Yaskawa INFORM job: DEMO_ROOF_UPPER_0625_3PAINT_48.JBI

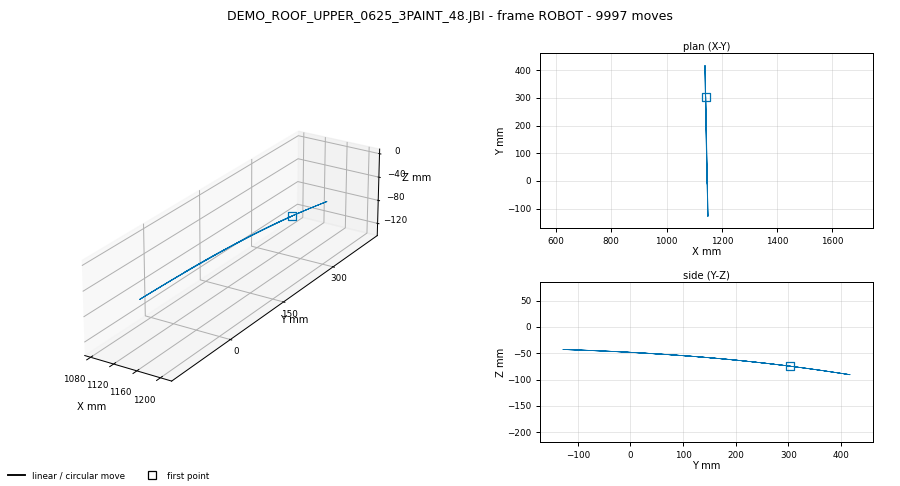
[picture p0: tool path of DEMO_ROOF_UPPER_0625_3PAINT_48.JBI in frame ROBOT, 9997 of 9997 moves have a stored position in this frame; points joined in program order, loops and branches not executed]
/JOB
//NAME DEMO_ROOF_UPPER_0625_3PAINT48
//POS
///NPOS 9997,0,0,0,0,0
///TOOL 0
///USER 0
///POSTYPE ROBOT
///RECTAN
///RCONF 1,0,0,0,0,0,0,0,0,0,0,0,0,0,0,0,0,0,0,0,0,0,0,0
C00000=1141.812,303.776,-74.472,-176.975,8.653,148.834
C00001=1141.816,303.528,-74.441,-176.978,8.649,148.834
C00002=1141.820,303.279,-74.410,-176.981,8.646,148.834
C00003=1141.824,303.032,-74.378,-176.983,8.643,148.834
C00004=1141.829,302.783,-74.347,-176.986,8.639,148.834
C00005=1141.833,302.536,-74.316,-176.989,8.636,148.834
C00006=1141.837,302.287,-74.285,-176.991,8.632,148.834
C00007=1141.841,302.040,-74.253,-176.994,8.628,148.833
C00008=1141.845,301.791,-74.222,-176.997,8.625,148.833
C00009=1141.849,301.544,-74.192,-177.000,8.621,148.833
C00010=1141.853,301.296,-74.160,-177.002,8.618,148.833
C00011=1141.857,301.048,-74.129,-177.005,8.615,148.833
C00012=1141.862,300.800,-74.099,-177.008,8.611,148.833
C00013=1141.866,300.552,-74.067,-177.010,8.608,148.833
C00014=1141.870,300.304,-74.036,-177.012,8.605,148.833
C00015=1141.874,300.055,-74.005,-177.016,8.601,148.833
C00016=1141.879,299.808,-73.973,-177.018,8.597,148.832
C00017=1141.883,299.559,-73.942,-177.020,8.594,148.832
C00018=1141.886,299.311,-73.912,-177.024,8.590,148.832
C00019=1141.891,299.063,-73.881,-177.026,8.587,148.832
C00020=1141.895,298.815,-73.849,-177.028,8.584,148.832
C00021=1141.899,298.567,-73.819,-177.032,8.580,148.832
C00022=1141.904,298.320,-73.788,-177.034,8.577,148.832
C00023=1141.907,298.071,-73.757,-177.036,8.574,148.832
C00024=1141.912,297.823,-73.727,-177.039,8.571,148.832
C00025=1141.916,297.575,-73.695,-177.042,8.567,148.831
C00026=1141.921,297.327,-73.665,-177.045,8.564,148.831
C00027=1141.925,297.079,-73.633,-177.047,8.560,148.831
C00028=1141.928,296.831,-73.603,-177.050,8.556,148.831
C00029=1141.933,296.583,-73.572,-177.053,8.553,148.831
C00030=1141.937,296.335,-73.541,-177.055,8.550,148.831
C00031=1141.941,296.087,-73.511,-177.058,8.546,148.831
C00032=1141.945,295.839,-73.480,-177.061,8.543,148.831
C00033=1141.950,295.591,-73.449,-177.063,8.540,148.831
C00034=1141.954,295.342,-73.418,-177.067,8.536,148.831
C00035=1141.958,295.094,-73.388,-177.069,8.533,148.830
C00036=1141.962,294.846,-73.357,-177.071,8.530,148.830
C00037=1141.966,294.598,-73.326,-177.074,8.527,148.830
C00038=1141.970,294.350,-73.296,-177.077,8.523,148.830
C00039=1141.975,294.102,-73.265,-177.080,8.520,148.830
C00040=1141.979,293.855,-73.235,-177.082,8.516,148.830
C00041=1141.983,293.606,-73.204,-177.085,8.512,148.830
C00042=1141.987,293.358,-73.173,-177.088,8.509,148.830
C00043=1141.991,293.110,-73.143,-177.090,8.506,148.830
C00044=1141.996,292.861,-73.112,-177.094,8.502,148.830
C00045=1141.999,292.613,-73.082,-177.096,8.499,148.829
C00046=1142.004,292.365,-73.051,-177.098,8.496,148.829
C00047=1142.009,292.117,-73.021,-177.101,8.493,148.829
C00048=1142.012,291.869,-72.990,-177.104,8.489,148.829
C00049=1142.017,291.621,-72.959,-177.107,8.486,148.829
C00050=1142.021,291.373,-72.930,-177.109,8.483,148.829
C00051=1142.025,291.125,-72.899,-177.112,8.480,148.829
C00052=1142.029,290.877,-72.869,-177.115,8.476,148.829
C00053=1142.033,290.629,-72.838,-177.118,8.473,148.829
C00054=1142.037,290.380,-72.808,-177.120,8.470,148.829
C00055=1142.042,290.132,-72.778,-177.123,8.466,148.829
C00056=1142.046,289.885,-72.747,-177.126,8.463,148.828
C00057=1142.051,289.636,-72.717,-177.128,8.459,148.828
C00058=1142.054,289.388,-72.687,-177.131,8.456,148.828
C00059=1142.059,289.140,-72.656,-177.134,8.452,148.828
C00060=1142.063,288.892,-72.627,-177.136,8.449,148.828
C00061=1142.067,288.644,-72.596,-177.139,8.446,148.828
C00062=1142.071,288.396,-72.566,-177.142,8.443,148.828
C00063=1142.076,288.147,-72.536,-177.144,8.439,148.828
C00064=1142.080,287.899,-72.505,-177.147,8.436,148.828
C00065=1142.084,287.624,-72.472,-177.150,8.432,148.828
C00066=1142.089,287.348,-72.438,-177.153,8.429,148.828
C00067=1142.094,287.073,-72.405,-177.156,8.425,148.828
C00068=1142.098,286.797,-72.372,-177.159,8.421,148.828
C00069=1142.103,286.549,-72.341,-177.162,8.418,148.828
C00070=1142.107,286.301,-72.312,-177.164,8.415,148.827
C00071=1142.111,286.053,-72.282,-177.167,8.412,148.827
C00072=1142.116,285.805,-72.252,-177.170,8.408,148.827
C00073=1142.120,285.557,-72.221,-177.173,8.405,148.827
C00074=1142.124,285.309,-72.192,-177.175,8.402,148.827
C00075=1142.129,285.061,-72.161,-177.178,8.399,148.827
C00076=1142.132,284.812,-72.131,-177.181,8.395,148.827
C00077=1142.136,284.563,-72.102,-177.184,8.392,148.827
C00078=1142.141,284.316,-72.071,-177.186,8.389,148.827
C00079=1142.145,284.067,-72.042,-177.189,8.386,148.827
C00080=1142.149,283.820,-72.011,-177.192,8.382,148.827
C00081=1142.154,283.571,-71.981,-177.194,8.379,148.827
C00082=1142.158,283.323,-71.952,-177.197,8.376,148.827
C00083=1142.162,283.075,-71.922,-177.200,8.373,148.827
C00084=1142.166,282.827,-71.892,-177.202,8.370,148.827
C00085=1142.171,282.578,-71.862,-177.205,8.366,148.826
C00086=1142.175,282.330,-71.833,-177.208,8.363,148.827
C00087=1142.179,282.082,-71.803,-177.210,8.359,148.826
C00088=1142.183,281.834,-71.773,-177.213,8.356,148.826
C00089=1142.187,281.586,-71.744,-177.217,8.353,148.826
C00090=1142.192,281.337,-71.714,-177.219,8.349,148.826
C00091=1142.196,281.090,-71.684,-177.222,8.347,148.826
C00092=1142.200,280.841,-71.654,-177.224,8.343,148.826
C00093=1142.205,280.593,-71.625,-177.227,8.340,148.826
C00094=1142.209,280.345,-71.595,-177.230,8.336,148.826
C00095=1142.213,280.097,-71.566,-177.233,8.333,148.826
C00096=1142.218,279.848,-71.536,-177.235,8.330,148.826
C00097=1142.222,279.600,-71.506,-177.238,8.327,148.826
C00098=1142.226,279.352,-71.476,-177.240,8.324,148.826
C00099=1142.230,279.104,-71.447,-177.244,8.320,148.826
C00100=1142.234,278.855,-71.417,-177.246,8.317,148.826
C00101=1142.239,278.607,-71.388,-177.249,8.314,148.826
C00102=1142.243,278.359,-71.358,-177.251,8.311,148.826
C00103=1142.247,278.111,-71.329,-177.254,8.308,148.826
C00104=1142.252,277.863,-71.300,-177.257,8.304,148.826
C00105=1142.256,277.615,-71.270,-177.260,8.301,148.826
C00106=1142.260,277.367,-71.241,-177.263,8.298,148.826
C00107=1142.264,277.118,-71.211,-177.265,8.295,148.826
C00108=1142.268,276.870,-71.182,-177.268,8.292,148.826
C00109=1142.273,276.622,-71.152,-177.270,8.289,148.826
C00110=1142.277,276.374,-71.123,-177.273,8.285,148.825
C00111=1142.281,276.125,-71.094,-177.276,8.282,148.825
C00112=1142.285,275.877,-71.064,-177.279,8.279,148.826
C00113=1142.290,275.628,-71.035,-177.281,8.276,148.825
C00114=1142.294,275.381,-71.006,-177.284,8.273,148.825
C00115=1142.299,275.132,-70.977,-177.287,8.270,148.825
C00116=1142.303,274.884,-70.947,-177.290,8.266,148.825
C00117=1142.307,274.636,-70.918,-177.293,8.263,148.825
C00118=1142.311,274.387,-70.888,-177.295,8.260,148.825
C00119=1142.315,274.139,-70.859,-177.298,8.257,148.825
C00120=1142.320,273.890,-70.830,-177.300,8.254,148.825
C00121=1142.325,273.643,-70.801,-177.303,8.251,148.825
C00122=1142.329,273.394,-70.772,-177.306,8.247,148.825
C00123=1142.332,273.147,-70.743,-177.309,8.244,148.825
C00124=1142.337,272.898,-70.714,-177.312,8.241,148.825
C00125=1142.341,272.649,-70.685,-177.314,8.238,148.825
C00126=1142.345,272.401,-70.655,-177.317,8.235,148.825
C00127=1142.350,272.153,-70.627,-177.320,8.232,148.825
C00128=1142.354,271.905,-70.597,-177.323,8.228,148.825
C00129=1142.358,271.656,-70.568,-177.325,8.225,148.825
C00130=1142.362,271.408,-70.540,-177.328,8.222,148.825
C00131=1142.367,271.160,-70.511,-177.331,8.219,148.825
C00132=1142.371,270.912,-70.481,-177.333,8.216,148.825
C00133=1142.376,270.663,-70.453,-177.336,8.213,148.825
C00134=1142.380,270.415,-70.423,-177.339,8.210,148.825
C00135=1142.383,270.167,-70.394,-177.342,8.206,148.825
C00136=1142.388,269.919,-70.366,-177.345,8.203,148.825
C00137=1142.393,269.670,-70.336,-177.347,8.200,148.825
C00138=1142.397,269.422,-70.308,-177.350,8.197,148.825
C00139=1142.401,269.174,-70.279,-177.353,8.194,148.825
C00140=1142.406,268.925,-70.250,-177.355,8.191,148.825
C00141=1142.410,268.677,-70.221,-177.358,8.188,148.825
C00142=1142.414,268.428,-70.192,-177.361,8.185,148.825
C00143=1142.418,268.181,-70.164,-177.364,8.181,148.825
C00144=1142.423,267.932,-70.135,-177.366,8.178,148.825
C00145=1142.427,267.684,-70.106,-177.369,8.175,148.825
C00146=1142.431,267.436,-70.078,-177.372,8.172,148.825
C00147=1142.436,267.187,-70.049,-177.374,8.169,148.825
C00148=1142.440,266.939,-70.020,-177.377,8.166,148.825
C00149=1142.444,266.691,-69.992,-177.380,8.163,148.825
C00150=1142.449,266.443,-69.962,-177.383,8.160,148.825
C00151=1142.453,266.194,-69.934,-177.386,8.157,148.825
C00152=1142.457,265.946,-69.906,-177.388,8.153,148.825
C00153=1142.462,265.698,-69.876,-177.391,8.150,148.825
C00154=1142.466,265.449,-69.848,-177.394,8.147,148.825
C00155=1142.470,265.201,-69.820,-177.397,8.144,148.825
C00156=1142.475,264.953,-69.790,-177.399,8.141,148.825
C00157=1142.478,264.704,-69.762,-177.402,8.138,148.825
C00158=1142.483,264.456,-69.734,-177.405,8.135,148.825
C00159=1142.488,264.207,-69.705,-177.408,8.132,148.825
C00160=1142.492,263.960,-69.677,-177.410,8.129,148.825
C00161=1142.496,263.711,-69.648,-177.413,8.125,148.825
C00162=1142.500,263.462,-69.620,-177.416,8.122,148.825
C00163=1142.505,263.214,-69.591,-177.419,8.119,148.825
C00164=1142.509,262.965,-69.563,-177.422,8.117,148.825
C00165=1142.514,262.718,-69.534,-177.424,8.114,148.825
C00166=1142.518,262.469,-69.506,-177.427,8.110,148.825
C00167=1142.522,262.220,-69.477,-177.430,8.107,148.825
C00168=1142.526,261.973,-69.450,-177.432,8.104,148.825
C00169=1142.532,261.699,-69.418,-177.436,8.101,148.825
C00170=1142.536,261.425,-69.387,-177.438,8.098,148.825
C00171=1142.541,261.152,-69.355,-177.442,8.094,148.825
C00172=1142.546,260.878,-69.325,-177.445,8.091,148.825
C00173=1142.549,260.630,-69.296,-177.447,8.088,148.825
C00174=1142.554,260.382,-69.268,-177.450,8.085,148.825
C00175=1142.558,260.133,-69.240,-177.453,8.082,148.825
C00176=1142.563,259.885,-69.211,-177.455,8.079,148.826
C00177=1142.567,259.636,-69.183,-177.458,8.076,148.826
C00178=1142.571,259.389,-69.156,-177.462,8.072,148.826
C00179=1142.576,259.140,-69.127,-177.464,8.070,148.826
C00180=1142.580,258.892,-69.099,-177.467,8.066,148.826
C00181=1142.585,258.643,-69.070,-177.469,8.063,148.826
C00182=1142.589,258.395,-69.043,-177.472,8.060,148.826
C00183=1142.593,258.146,-69.014,-177.475,8.058,148.826
C00184=1142.598,257.898,-68.986,-177.478,8.055,148.826
C00185=1142.602,257.649,-68.959,-177.481,8.052,148.826
C00186=1142.606,257.401,-68.931,-177.483,8.049,148.826
C00187=1142.611,257.152,-68.902,-177.486,8.045,148.826
C00188=1142.615,256.904,-68.874,-177.488,8.043,148.826
C00189=1142.619,256.656,-68.846,-177.491,8.040,148.826
C00190=1142.623,256.408,-68.818,-177.494,8.037,148.826
C00191=1142.628,256.159,-68.790,-177.497,8.034,148.826
C00192=1142.632,255.911,-68.763,-177.500,8.031,148.826
C00193=1142.637,255.663,-68.735,-177.502,8.028,148.826
C00194=1142.641,255.414,-68.706,-177.505,8.025,148.826
C00195=1142.646,255.166,-68.678,-177.508,8.022,148.826
C00196=1142.650,254.917,-68.651,-177.510,8.019,148.826
C00197=1142.654,254.669,-68.623,-177.514,8.015,148.826
C00198=1142.658,254.420,-68.595,-177.517,8.012,148.826
C00199=1142.663,254.171,-68.567,-177.519,8.009,148.826
C00200=1142.667,253.924,-68.540,-177.522,8.006,148.826
C00201=1142.671,253.675,-68.511,-177.525,8.003,148.826
C00202=1142.676,253.426,-68.484,-177.528,8.000,148.827
C00203=1142.680,253.179,-68.457,-177.530,7.998,148.827
C00204=1142.685,252.930,-68.428,-177.533,7.995,148.827
C00205=1142.689,252.681,-68.401,-177.536,7.991,148.827
C00206=1142.693,252.433,-68.373,-177.538,7.988,148.827
C00207=1142.697,252.185,-68.345,-177.541,7.986,148.827
C00208=1142.702,251.936,-68.318,-177.544,7.983,148.827
C00209=1142.706,251.688,-68.290,-177.547,7.980,148.827
C00210=1142.711,251.439,-68.263,-177.550,7.977,148.827
C00211=1142.715,251.191,-68.235,-177.552,7.974,148.827
C00212=1142.719,250.942,-68.207,-177.555,7.971,148.827
C00213=1142.724,250.694,-68.179,-177.558,7.968,148.827
C00214=1142.729,250.445,-68.152,-177.561,7.965,148.827
C00215=1142.732,250.197,-68.124,-177.564,7.962,148.827
C00216=1142.737,249.948,-68.097,-177.566,7.959,148.827
C00217=1142.741,249.701,-68.069,-177.569,7.956,148.827
C00218=1142.746,249.451,-68.042,-177.572,7.953,148.827
C00219=1142.750,249.203,-68.014,-177.574,7.950,148.827
C00220=1142.755,248.955,-67.987,-177.577,7.947,148.827
C00221=1142.759,248.706,-67.960,-177.580,7.944,148.827
C00222=1142.763,248.458,-67.931,-177.583,7.941,148.828
C00223=1142.768,248.209,-67.904,-177.585,7.938,148.828
C00224=1142.772,247.961,-67.877,-177.588,7.936,148.828
C00225=1142.777,247.713,-67.850,-177.591,7.933,148.828
C00226=1142.781,247.464,-67.822,-177.594,7.930,148.828
C00227=1142.785,247.215,-67.795,-177.597,7.927,148.828
C00228=1142.790,246.967,-67.767,-177.599,7.924,148.828
C00229=1142.794,246.719,-67.740,-177.602,7.921,148.828
C00230=1142.798,246.470,-67.713,-177.605,7.918,148.828
C00231=1142.803,246.221,-67.686,-177.608,7.915,148.828
C00232=1142.807,245.974,-67.659,-177.611,7.912,148.828
C00233=1142.811,245.725,-67.632,-177.613,7.909,148.828
C00234=1142.815,245.476,-67.604,-177.616,7.906,148.828
C00235=1142.820,245.227,-67.577,-177.619,7.903,148.829
C00236=1142.824,244.980,-67.549,-177.622,7.900,148.829
C00237=1142.829,244.731,-67.522,-177.625,7.898,148.829
C00238=1142.834,244.483,-67.495,-177.627,7.895,148.829
C00239=1142.838,244.234,-67.468,-177.630,7.892,148.829
C00240=1142.842,243.985,-67.441,-177.633,7.889,148.829
C00241=1142.846,243.737,-67.414,-177.635,7.887,148.829
C00242=1142.851,243.488,-67.387,-177.638,7.884,148.829
C00243=1142.855,243.240,-67.359,-177.641,7.881,148.829
C00244=1142.860,242.992,-67.332,-177.643,7.878,148.829
C00245=1142.865,242.743,-67.305,-177.646,7.875,148.829
C00246=1142.868,242.495,-67.278,-177.649,7.872,148.829
C00247=1142.873,242.246,-67.251,-177.652,7.869,148.829
C00248=1142.877,241.998,-67.224,-177.655,7.866,148.830
C00249=1142.882,241.749,-67.197,-177.657,7.863,148.830
C00250=1142.886,241.501,-67.171,-177.660,7.860,148.830
C00251=1142.890,241.252,-67.144,-177.663,7.858,148.830
C00252=1142.895,241.004,-67.117,-177.666,7.855,148.830
C00253=1142.900,240.755,-67.090,-177.669,7.852,148.830
C00254=1142.903,240.506,-67.063,-177.671,7.849,148.830
C00255=1142.908,240.258,-67.036,-177.674,7.846,148.830
C00256=1142.912,240.009,-67.009,-177.677,7.843,148.830
C00257=1142.917,239.761,-66.983,-177.680,7.840,148.830
C00258=1142.921,239.512,-66.956,-177.683,7.837,148.830
C00259=1142.926,239.264,-66.929,-177.685,7.834,148.830
C00260=1142.930,239.015,-66.902,-177.688,7.832,148.831
C00261=1142.935,238.767,-66.875,-177.691,7.829,148.831
C00262=1142.939,238.519,-66.848,-177.694,7.827,148.831
C00263=1142.943,238.270,-66.822,-177.696,7.824,148.831
C00264=1142.948,238.021,-66.795,-177.699,7.821,148.831
C00265=1142.953,237.773,-66.768,-177.702,7.818,148.831
C00266=1142.957,237.525,-66.742,-177.705,7.815,148.831
C00267=1142.961,237.276,-66.715,-177.708,7.812,148.831
C00268=1142.966,237.028,-66.688,-177.710,7.809,148.831
C00269=1142.970,236.779,-66.662,-177.713,7.806,148.831
C00270=1142.975,236.530,-66.635,-177.716,7.803,148.832
C00271=1142.979,236.282,-66.608,-177.719,7.800,148.832
C00272=1142.984,236.033,-66.582,-177.721,7.798,148.832
C00273=1142.988,235.761,-66.552,-177.724,7.794,148.832
C00274=1142.993,235.489,-66.524,-177.728,7.792,148.832
C00275=1142.998,235.218,-66.494,-177.730,7.789,148.832
C00276=1143.003,234.946,-66.466,-177.734,7.785,148.832
C00277=1143.007,234.697,-66.439,-177.736,7.783,148.832
C00278=1143.012,234.448,-66.413,-177.739,7.780,148.832
C00279=1143.016,234.200,-66.386,-177.742,7.777,148.832
C00280=1143.021,233.952,-66.359,-177.744,7.774,148.833
C00281=1143.025,233.703,-66.333,-177.747,7.771,148.833
C00282=1143.030,233.454,-66.306,-177.750,7.769,148.833
C00283=1143.034,233.205,-66.281,-177.753,7.766,148.833
C00284=1143.038,232.957,-66.254,-177.756,7.763,148.833
C00285=1143.043,232.708,-66.228,-177.759,7.760,148.833
C00286=1143.047,232.460,-66.201,-177.762,7.757,148.833
C00287=1143.052,232.211,-66.175,-177.764,7.755,148.833
C00288=1143.055,231.963,-66.149,-177.767,7.752,148.834
C00289=1143.060,231.714,-66.122,-177.769,7.749,148.834
C00290=1143.064,231.465,-66.096,-177.772,7.746,148.834
C00291=1143.069,231.217,-66.070,-177.776,7.744,148.834
C00292=1143.074,230.969,-66.043,-177.778,7.741,148.834
C00293=1143.078,230.720,-66.018,-177.781,7.738,148.834
C00294=1143.083,230.471,-65.991,-177.784,7.735,148.834
C00295=1143.087,230.223,-65.965,-177.786,7.733,148.834
C00296=1143.091,229.974,-65.939,-177.789,7.730,148.834
C00297=1143.096,229.725,-65.912,-177.792,7.727,148.835
C00298=1143.100,229.477,-65.886,-177.795,7.724,148.835
C00299=1143.105,229.228,-65.861,-177.798,7.722,148.835
C00300=1143.110,228.980,-65.834,-177.801,7.719,148.835
C00301=1143.114,228.731,-65.808,-177.803,7.716,148.835
C00302=1143.118,228.482,-65.782,-177.806,7.714,148.835
C00303=1143.122,228.234,-65.756,-177.808,7.711,148.835
C00304=1143.127,227.985,-65.729,-177.811,7.708,148.835
C00305=1143.131,227.736,-65.704,-177.814,7.705,148.835
C00306=1143.136,227.488,-65.678,-177.817,7.702,148.836
C00307=1143.141,227.240,-65.651,-177.820,7.700,148.836
C00308=1143.145,226.991,-65.625,-177.823,7.697,148.836
C00309=1143.149,226.742,-65.600,-177.825,7.694,148.836
C00310=1143.153,226.493,-65.574,-177.828,7.692,148.836
C00311=1143.158,226.245,-65.549,-177.831,7.689,148.836
C00312=1143.163,225.997,-65.522,-177.834,7.686,148.837
C00313=1143.167,225.748,-65.496,-177.837,7.683,148.837
C00314=1143.171,225.499,-65.470,-177.840,7.680,148.837
C00315=1143.176,225.251,-65.445,-177.842,7.678,148.837
C00316=1143.180,225.002,-65.419,-177.845,7.675,148.837
C00317=1143.185,224.753,-65.393,-177.848,7.673,148.837
C00318=1143.189,224.504,-65.367,-177.851,7.670,148.837
C00319=1143.194,224.256,-65.341,-177.853,7.667,148.837
C00320=1143.198,224.007,-65.316,-177.856,7.664,148.838
C00321=1143.202,223.759,-65.289,-177.858,7.662,148.838
C00322=1143.207,223.510,-65.263,-177.861,7.659,148.838
C00323=1143.211,223.262,-65.238,-177.864,7.656,148.838
C00324=1143.216,223.013,-65.212,-177.867,7.653,148.838
C00325=1143.221,222.764,-65.186,-177.870,7.651,148.838
C00326=1143.225,222.515,-65.160,-177.872,7.648,148.838
C00327=1143.230,222.267,-65.135,-177.876,7.646,148.839
C00328=1143.234,222.019,-65.109,-177.878,7.643,148.839
C00329=1143.238,221.769,-65.084,-177.881,7.640,148.839
C00330=1143.243,221.521,-65.059,-177.884,7.637,148.839
C00331=1143.247,221.272,-65.033,-177.886,7.635,148.839
C00332=1143.252,221.023,-65.007,-177.889,7.632,148.839
C00333=1143.257,220.775,-64.982,-177.892,7.630,148.839
C00334=1143.261,220.527,-64.956,-177.895,7.627,148.840
C00335=1143.265,220.278,-64.930,-177.898,7.624,148.840
C00336=1143.270,220.030,-64.905,-177.900,7.622,148.840
C00337=1143.274,219.781,-64.879,-177.903,7.619,148.840
C00338=1143.279,219.531,-64.854,-177.906,7.616,148.840
C00339=1143.283,219.283,-64.829,-177.909,7.613,148.840
C00340=1143.288,219.034,-64.803,-177.912,7.610,148.840
C00341=1143.292,218.786,-64.777,-177.914,7.609,148.841
C00342=1143.297,218.538,-64.752,-177.917,7.606,148.841
C00343=1143.301,218.288,-64.727,-177.920,7.603,148.841
C00344=1143.306,218.040,-64.701,-177.923,7.600,148.841
C00345=1143.310,217.791,-64.676,-177.925,7.598,148.841
C00346=1143.314,217.542,-64.650,-177.928,7.595,148.841
C00347=1143.320,217.294,-64.625,-177.931,7.592,148.842
C00348=1143.323,217.045,-64.600,-177.934,7.589,148.842
C00349=1143.328,216.797,-64.575,-177.937,7.587,148.842
C00350=1143.332,216.548,-64.550,-177.939,7.585,148.842
C00351=1143.337,216.299,-64.524,-177.942,7.582,148.842
C00352=1143.341,216.051,-64.499,-177.945,7.579,148.842
C00353=1143.346,215.801,-64.473,-177.948,7.576,148.843
C00354=1143.351,215.553,-64.448,-177.950,7.574,148.843
C00355=1143.355,215.304,-64.424,-177.953,7.571,148.843
C00356=1143.359,215.056,-64.398,-177.956,7.569,148.843
C00357=1143.364,214.807,-64.373,-177.959,7.566,148.843
C00358=1143.369,214.558,-64.348,-177.962,7.564,148.843
C00359=1143.373,214.310,-64.322,-177.964,7.561,148.843
C00360=1143.378,214.060,-64.297,-177.968,7.558,148.844
C00361=1143.382,213.812,-64.272,-177.970,7.555,148.844
C00362=1143.386,213.563,-64.247,-177.973,7.553,148.844
C00363=1143.391,213.315,-64.222,-177.976,7.551,148.844
C00364=1143.396,213.066,-64.197,-177.979,7.548,148.844
C00365=1143.400,212.818,-64.172,-177.981,7.545,148.844
C00366=1143.404,212.568,-64.147,-177.984,7.543,148.845
C00367=1143.409,212.320,-64.122,-177.987,7.540,148.845
C00368=1143.414,212.071,-64.097,-177.990,7.537,148.845
C00369=1143.418,211.823,-64.072,-177.992,7.535,148.845
C00370=1143.423,211.574,-64.047,-177.995,7.533,148.845
C00371=1143.427,211.325,-64.022,-177.998,7.530,148.846
C00372=1143.431,211.077,-63.997,-178.001,7.527,148.846
C00373=1143.436,210.828,-63.972,-178.004,7.525,148.846
C00374=1143.441,210.580,-63.947,-178.006,7.522,148.846
C00375=1143.444,210.330,-63.922,-178.009,7.519,148.846
C00376=1143.450,210.082,-63.898,-178.012,7.517,148.847
C00377=1143.454,209.811,-63.871,-178.015,7.514,148.847
C00378=1143.459,209.541,-63.844,-178.018,7.511,148.847
C00379=1143.465,209.269,-63.816,-178.021,7.508,148.847
C00380=1143.470,208.999,-63.790,-178.025,7.506,148.847
C00381=1143.474,208.750,-63.765,-178.027,7.504,148.847
C00382=1143.478,208.502,-63.740,-178.030,7.501,148.848
C00383=1143.483,208.253,-63.715,-178.033,7.498,148.848
C00384=1143.487,208.004,-63.691,-178.035,7.496,148.848
C00385=1143.492,207.755,-63.666,-178.038,7.493,148.848
C00386=1143.496,207.507,-63.641,-178.041,7.491,148.848
C00387=1143.501,207.258,-63.616,-178.044,7.488,148.849
C00388=1143.505,207.009,-63.592,-178.046,7.486,148.849
C00389=1143.510,206.760,-63.567,-178.049,7.483,148.849
C00390=1143.515,206.512,-63.542,-178.052,7.480,148.849
C00391=1143.519,206.263,-63.518,-178.054,7.478,148.849
C00392=1143.524,206.014,-63.493,-178.058,7.475,148.850
C00393=1143.528,205.766,-63.468,-178.061,7.473,148.850
C00394=1143.533,205.517,-63.443,-178.063,7.471,148.850
C00395=1143.537,205.268,-63.419,-178.066,7.468,148.850
C00396=1143.542,205.020,-63.395,-178.069,7.465,148.850
C00397=1143.546,204.770,-63.370,-178.071,7.463,148.851
C00398=1143.551,204.522,-63.346,-178.074,7.460,148.851
C00399=1143.556,204.273,-63.322,-178.078,7.458,148.851
C00400=1143.560,204.024,-63.296,-178.080,7.456,148.851
C00401=1143.564,203.775,-63.272,-178.083,7.453,148.851
C00402=1143.569,203.527,-63.248,-178.086,7.450,148.852
C00403=1143.574,203.278,-63.224,-178.088,7.448,148.852
C00404=1143.578,203.029,-63.199,-178.091,7.446,148.852
C00405=1143.583,202.780,-63.175,-178.094,7.443,148.852
C00406=1143.587,202.532,-63.150,-178.096,7.441,148.852
C00407=1143.591,202.283,-63.126,-178.100,7.438,148.853
C00408=1143.596,202.034,-63.101,-178.102,7.435,148.853
C00409=1143.601,201.786,-63.077,-178.105,7.433,148.853
C00410=1143.606,201.537,-63.053,-178.108,7.430,148.853
C00411=1143.610,201.287,-63.029,-178.110,7.428,148.853
C00412=1143.614,201.039,-63.005,-178.113,7.426,148.854
C00413=1143.619,200.790,-62.980,-178.116,7.423,148.854
C00414=1143.624,200.542,-62.956,-178.119,7.421,148.854
C00415=1143.628,200.293,-62.932,-178.122,7.418,148.854
C00416=1143.633,200.044,-62.907,-178.125,7.416,148.854
C00417=1143.637,199.795,-62.884,-178.127,7.414,148.855
C00418=1143.642,199.547,-62.860,-178.130,7.411,148.855
C00419=1143.646,199.297,-62.835,-178.133,7.408,148.855
C00420=1143.651,199.049,-62.810,-178.136,7.406,148.855
C00421=1143.655,198.800,-62.786,-178.139,7.404,148.856
C00422=1143.660,198.551,-62.763,-178.141,7.401,148.856
C00423=1143.665,198.303,-62.738,-178.144,7.399,148.856
C00424=1143.669,198.054,-62.714,-178.147,7.396,148.856
C00425=1143.673,197.804,-62.691,-178.150,7.394,148.856
C00426=1143.678,197.556,-62.666,-178.153,7.391,148.857
C00427=1143.683,197.307,-62.642,-178.155,7.388,148.857
C00428=1143.688,197.058,-62.618,-178.158,7.387,148.857
C00429=1143.692,196.810,-62.594,-178.161,7.384,148.857
C00430=1143.696,196.561,-62.570,-178.164,7.382,148.857
C00431=1143.701,196.312,-62.547,-178.166,7.379,148.858
C00432=1143.706,196.063,-62.522,-178.170,7.377,148.858
C00433=1143.710,195.814,-62.498,-178.172,7.375,148.858
C00434=1143.715,195.565,-62.474,-178.175,7.372,148.858
C00435=1143.719,195.317,-62.450,-178.177,7.370,148.859
C00436=1143.724,195.068,-62.427,-178.181,7.367,148.859
C00437=1143.728,194.820,-62.403,-178.183,7.364,148.859
C00438=1143.732,194.570,-62.379,-178.186,7.363,148.859
C00439=1143.737,194.321,-62.355,-178.189,7.360,148.859
C00440=1143.742,194.072,-62.331,-178.192,7.358,148.860
C00441=1143.747,193.824,-62.307,-178.194,7.355,148.860
C00442=1143.751,193.575,-62.284,-178.197,7.353,148.860
C00443=1143.756,193.326,-62.260,-178.200,7.350,148.860
C00444=1143.760,193.077,-62.236,-178.203,7.348,148.861
C00445=1143.765,192.829,-62.212,-178.205,7.346,148.861
C00446=1143.769,192.580,-62.189,-178.209,7.343,148.861
C00447=1143.774,192.331,-62.165,-178.211,7.341,148.861
C00448=1143.779,192.082,-62.141,-178.214,7.339,148.862
C00449=1143.783,191.834,-62.117,-178.216,7.337,148.862
C00450=1143.788,191.585,-62.094,-178.220,7.334,148.862
C00451=1143.793,191.336,-62.070,-178.223,7.331,148.862
C00452=1143.797,191.087,-62.046,-178.225,7.329,148.863
C00453=1143.802,190.838,-62.023,-178.228,7.326,148.863
C00454=1143.807,190.589,-61.999,-178.231,7.325,148.863
C00455=1143.811,190.340,-61.975,-178.234,7.322,148.863
C00456=1143.815,190.091,-61.951,-178.236,7.320,148.864
C00457=1143.820,189.842,-61.928,-178.239,7.317,148.864
C00458=1143.824,189.593,-61.904,-178.242,7.315,148.864
C00459=1143.828,189.345,-61.881,-178.245,7.313,148.864
C00460=1143.834,189.096,-61.858,-178.248,7.310,148.864
C00461=1143.838,188.847,-61.835,-178.251,7.308,148.865
C00462=1143.843,188.599,-61.811,-178.253,7.305,148.865
C00463=1143.848,188.350,-61.787,-178.256,7.304,148.865
C00464=1143.852,188.101,-61.764,-178.259,7.301,148.865
C00465=1143.857,187.852,-61.741,-178.262,7.299,148.866
C00466=1143.862,187.603,-61.717,-178.264,7.296,148.866
C00467=1143.866,187.354,-61.693,-178.267,7.294,148.866
C00468=1143.871,187.105,-61.670,-178.270,7.291,148.866
C00469=1143.875,186.856,-61.647,-178.273,7.290,148.867
C00470=1143.880,186.607,-61.623,-178.276,7.287,148.867
C00471=1143.884,186.359,-61.600,-178.278,7.285,148.867
C00472=1143.889,186.110,-61.577,-178.281,7.283,148.868
C00473=1143.893,185.861,-61.554,-178.284,7.280,148.868
C00474=1143.898,185.612,-61.530,-178.287,7.278,148.868
C00475=1143.903,185.362,-61.507,-178.290,7.275,148.868
C00476=1143.907,185.114,-61.483,-178.292,7.273,148.869
C00477=1143.911,184.865,-61.460,-178.295,7.270,148.869
C00478=1143.917,184.617,-61.437,-178.298,7.269,148.869
C00479=1143.921,184.368,-61.414,-178.301,7.266,148.869
C00480=1143.926,184.119,-61.391,-178.303,7.264,148.869
C00481=1143.931,183.849,-61.365,-178.307,7.261,148.870
C00482=1143.936,183.580,-61.341,-178.310,7.259,148.870
C00483=1143.941,183.309,-61.316,-178.313,7.256,148.870
C00484=1143.946,183.040,-61.290,-178.315,7.254,148.871
C00485=1143.951,182.790,-61.267,-178.319,7.252,148.871
C00486=1143.955,182.542,-61.245,-178.321,7.250,148.871
C00487=1143.960,182.293,-61.221,-178.324,7.247,148.871
C00488=1143.965,182.044,-61.198,-178.327,7.245,148.872
C00489=1143.968,181.796,-61.175,-178.330,7.242,148.872
C00490=1143.973,181.547,-61.152,-178.332,7.241,148.872
C00491=1143.978,181.298,-61.129,-178.335,7.238,148.872
C00492=1143.982,181.049,-61.106,-178.338,7.236,148.873
C00493=1143.987,180.801,-61.083,-178.341,7.234,148.873
C00494=1143.992,180.551,-61.060,-178.343,7.231,148.873
C00495=1143.996,180.302,-61.037,-178.347,7.229,148.874
C00496=1144.001,180.053,-61.014,-178.349,7.227,148.874
C00497=1144.006,179.804,-60.991,-178.352,7.224,148.874
C00498=1144.010,179.556,-60.968,-178.355,7.223,148.874
C00499=1144.015,179.306,-60.946,-178.358,7.220,148.875
C00500=1144.020,179.057,-60.922,-178.360,7.218,148.875
C00501=1144.024,178.809,-60.900,-178.363,7.216,148.875
C00502=1144.028,178.560,-60.876,-178.366,7.213,148.875
C00503=1144.033,178.311,-60.855,-178.369,7.212,148.876
C00504=1144.038,178.062,-60.831,-178.371,7.209,148.876
C00505=1144.043,177.813,-60.808,-178.374,7.207,148.876
C00506=1144.047,177.564,-60.785,-178.377,7.204,148.877
C00507=1144.052,177.315,-60.763,-178.380,7.202,148.877
C00508=1144.056,177.067,-60.740,-178.383,7.200,148.877
C00509=1144.061,176.818,-60.717,-178.386,7.198,148.878
C00510=1144.065,176.568,-60.695,-178.388,7.195,148.878
C00511=1144.071,176.320,-60.672,-178.391,7.193,148.878
C00512=1144.075,176.071,-60.650,-178.394,7.192,148.878
C00513=1144.079,175.821,-60.626,-178.397,7.189,148.879
C00514=1144.084,175.573,-60.604,-178.399,7.187,148.879
C00515=1144.089,175.324,-60.581,-178.403,7.185,148.879
C00516=1144.093,175.075,-60.558,-178.405,7.182,148.879
C00517=1144.098,174.825,-60.536,-178.408,7.180,148.880
C00518=1144.103,174.577,-60.513,-178.411,7.178,148.880
C00519=1144.108,174.328,-60.491,-178.414,7.175,148.880
C00520=1144.112,174.079,-60.468,-178.416,7.174,148.881
C00521=1144.117,173.830,-60.446,-178.419,7.172,148.881
C00522=1144.121,173.581,-60.423,-178.422,7.169,148.881
C00523=1144.125,173.332,-60.401,-178.425,7.167,148.881
C00524=1144.131,173.084,-60.378,-178.428,7.165,148.882
C00525=1144.135,172.834,-60.356,-178.430,7.163,148.882
C00526=1144.140,172.585,-60.332,-178.433,7.161,148.882
C00527=1144.145,172.337,-60.311,-178.436,7.158,148.883
C00528=1144.149,172.088,-60.287,-178.438,7.156,148.883
C00529=1144.154,171.839,-60.266,-178.442,7.154,148.883
C00530=1144.158,171.590,-60.244,-178.444,7.152,148.884
C00531=1144.163,171.341,-60.220,-178.448,7.149,148.884
C00532=1144.168,171.092,-60.199,-178.450,7.147,148.884
C00533=1144.172,170.843,-60.176,-178.453,7.146,148.884
C00534=1144.177,170.594,-60.154,-178.456,7.143,148.885
C00535=1144.182,170.345,-60.132,-178.458,7.141,148.885
C00536=1144.186,170.096,-60.109,-178.461,7.138,148.885
C00537=1144.191,169.847,-60.087,-178.464,7.137,148.886
C00538=1144.196,169.598,-60.064,-178.466,7.135,148.886
C00539=1144.200,169.349,-60.043,-178.470,7.132,148.886
C00540=1144.205,169.100,-60.019,-178.472,7.130,148.887
C00541=1144.209,168.851,-59.997,-178.476,7.128,148.887
C00542=1144.214,168.602,-59.976,-178.478,7.126,148.887
C00543=1144.219,168.353,-59.954,-178.480,7.124,148.887
C00544=1144.224,168.105,-59.931,-178.484,7.121,148.888
C00545=1144.228,167.855,-59.909,-178.486,7.120,148.888
C00546=1144.233,167.607,-59.887,-178.489,7.118,148.888
C00547=1144.238,167.357,-59.864,-178.492,7.115,148.889
C00548=1144.243,167.108,-59.843,-178.495,7.113,148.889
C00549=1144.247,166.860,-59.820,-178.498,7.111,148.889
C00550=1144.252,166.611,-59.798,-178.500,7.109,148.889
C00551=1144.256,166.362,-59.776,-178.503,7.107,148.890
C00552=1144.262,166.113,-59.754,-178.506,7.105,148.890
C00553=1144.266,165.863,-59.732,-178.508,7.102,148.890
C00554=1144.271,165.615,-59.710,-178.511,7.101,148.891
C00555=1144.275,165.365,-59.688,-178.514,7.098,148.891
C00556=1144.280,165.117,-59.666,-178.517,7.096,148.891
C00557=1144.284,164.868,-59.644,-178.519,7.094,148.892
C00558=1144.289,164.619,-59.621,-178.523,7.092,148.892
C00559=1144.294,164.370,-59.599,-178.525,7.090,148.892
C00560=1144.299,164.121,-59.578,-178.528,7.088,148.893
C00561=1144.303,163.872,-59.556,-178.531,7.086,148.893
C00562=1144.308,163.623,-59.534,-178.534,7.084,148.893
C00563=1144.312,163.374,-59.512,-178.537,7.081,148.894
C00564=1144.317,163.125,-59.490,-178.540,7.080,148.894
C00565=1144.321,162.876,-59.468,-178.542,7.077,148.894
C00566=1144.326,162.627,-59.446,-178.545,7.075,148.894
C00567=1144.330,162.378,-59.424,-178.548,7.073,148.895
C00568=1144.336,162.129,-59.402,-178.551,7.071,148.895
C00569=1144.341,161.880,-59.381,-178.554,7.069,148.896
C00570=1144.345,161.630,-59.359,-178.556,7.067,148.896
C00571=1144.350,161.382,-59.337,-178.559,7.065,148.896
C00572=1144.354,161.132,-59.315,-178.562,7.063,148.896
C00573=1144.359,160.884,-59.294,-178.565,7.061,148.897
C00574=1144.364,160.634,-59.272,-178.567,7.059,148.897
C00575=1144.368,160.386,-59.250,-178.570,7.057,148.897
C00576=1144.373,160.137,-59.228,-178.573,7.055,148.898
C00577=1144.378,159.887,-59.207,-178.576,7.053,148.898
C00578=1144.383,159.638,-59.185,-178.578,7.051,148.899
C00579=1144.388,159.390,-59.164,-178.581,7.048,148.899
C00580=1144.392,159.140,-59.142,-178.584,7.047,148.899
C00581=1144.397,158.892,-59.120,-178.587,7.045,148.899
C00582=1144.401,158.642,-59.098,-178.590,7.042,148.900
C00583=1144.406,158.393,-59.077,-178.593,7.041,148.900
C00584=1144.410,158.145,-59.056,-178.595,7.038,148.900
C00585=1144.416,157.876,-59.032,-178.598,7.036,148.901
C00586=1144.421,157.607,-59.008,-178.601,7.034,148.901
C00587=1144.426,157.338,-58.986,-178.604,7.032,148.901
C00588=1144.431,157.068,-58.962,-178.607,7.029,148.902
C00589=1144.435,156.820,-58.941,-178.610,7.027,148.902
C00590=1144.440,156.571,-58.919,-178.613,7.026,148.903
C00591=1144.445,156.321,-58.898,-178.616,7.024,148.903
C00592=1144.450,156.073,-58.876,-178.618,7.021,148.903
C00593=1144.454,155.823,-58.854,-178.621,7.019,148.903
C00594=1144.459,155.574,-58.833,-178.624,7.018,148.904
C00595=1144.464,155.326,-58.812,-178.627,7.015,148.904
C00596=1144.469,155.076,-58.791,-178.630,7.013,148.905
C00597=1144.473,154.827,-58.769,-178.633,7.012,148.905
C00598=1144.478,154.579,-58.748,-178.635,7.010,148.905
C00599=1144.483,154.329,-58.727,-178.638,7.007,148.905
C00600=1144.487,154.080,-58.705,-178.641,7.005,148.906
C00601=1144.492,153.831,-58.684,-178.643,7.004,148.906
C00602=1144.496,153.582,-58.663,-178.646,7.002,148.907
C00603=1144.501,153.333,-58.642,-178.649,6.999,148.907
C00604=1144.506,153.084,-58.620,-178.652,6.997,148.907
C00605=1144.511,152.835,-58.599,-178.654,6.996,148.907
C00606=1144.516,152.586,-58.577,-178.658,6.993,148.908
C00607=1144.520,152.337,-58.556,-178.660,6.991,148.908
C00608=1144.525,152.088,-58.535,-178.663,6.990,148.909
C00609=1144.530,151.838,-58.513,-178.666,6.988,148.909
C00610=1144.535,151.590,-58.492,-178.669,6.985,148.909
C00611=1144.539,151.341,-58.471,-178.671,6.983,148.910
C00612=1144.544,151.092,-58.450,-178.674,6.982,148.910
C00613=1144.549,150.843,-58.429,-178.677,6.980,148.910
C00614=1144.553,150.593,-58.408,-178.680,6.977,148.911
C00615=1144.558,150.345,-58.386,-178.683,6.976,148.911
C00616=1144.563,150.095,-58.365,-178.686,6.974,148.911
C00617=1144.567,149.846,-58.345,-178.688,6.972,148.912
C00618=1144.572,149.598,-58.323,-178.690,6.970,148.912
C00619=1144.577,149.348,-58.302,-178.694,6.968,148.912
C00620=1144.581,149.099,-58.282,-178.696,6.966,148.913
C00621=1144.586,148.850,-58.260,-178.699,6.964,148.913
C00622=1144.591,148.601,-58.239,-178.702,6.963,148.914
C00623=1144.596,148.352,-58.219,-178.705,6.960,148.914
C00624=1144.601,148.103,-58.198,-178.708,6.958,148.914
C00625=1144.606,147.854,-58.176,-178.711,6.957,148.915
C00626=1144.610,147.604,-58.155,-178.713,6.955,148.915
C00627=1144.615,147.355,-58.134,-178.716,6.952,148.915
C00628=1144.619,147.106,-58.114,-178.719,6.950,148.916
C00629=1144.624,146.858,-58.092,-178.722,6.949,148.916
C00630=1144.629,146.608,-58.071,-178.724,6.947,148.916
C00631=1144.634,146.359,-58.051,-178.727,6.945,148.917
C00632=1144.639,146.110,-58.030,-178.730,6.943,148.917
C00633=1144.643,145.861,-58.010,-178.733,6.941,148.917
C00634=1144.648,145.612,-57.989,-178.736,6.939,148.918
C00635=1144.652,145.363,-57.967,-178.738,6.937,148.918
C00636=1144.657,145.114,-57.946,-178.741,6.935,148.918
C00637=1144.662,144.865,-57.926,-178.744,6.933,148.919
C00638=1144.667,144.615,-57.905,-178.747,6.931,148.919
C00639=1144.671,144.366,-57.884,-178.749,6.929,148.920
C00640=1144.676,144.117,-57.863,-178.752,6.928,148.920
C00641=1144.681,143.868,-57.843,-178.755,6.926,148.920
C00642=1144.686,143.619,-57.822,-178.758,6.924,148.921
C00643=1144.690,143.370,-57.802,-178.761,6.922,148.921
C00644=1144.696,143.121,-57.781,-178.764,6.920,148.921
C00645=1144.700,142.872,-57.760,-178.766,6.918,148.922
C00646=1144.705,142.623,-57.739,-178.769,6.917,148.922
C00647=1144.710,142.374,-57.719,-178.772,6.915,148.923
C00648=1144.714,142.125,-57.699,-178.775,6.912,148.923
C00649=1144.719,141.875,-57.678,-178.777,6.910,148.923
C00650=1144.724,141.626,-57.657,-178.780,6.909,148.924
C00651=1144.729,141.377,-57.636,-178.783,6.907,148.924
C00652=1144.733,141.128,-57.616,-178.785,6.905,148.924
C00653=1144.738,140.879,-57.596,-178.789,6.903,148.925
C00654=1144.743,140.630,-57.575,-178.791,6.901,148.925
C00655=1144.747,140.381,-57.554,-178.794,6.899,148.926
C00656=1144.753,140.132,-57.533,-178.797,6.898,148.926
C00657=1144.757,139.883,-57.513,-178.800,6.896,148.926
C00658=1144.761,139.634,-57.493,-178.802,6.894,148.927
C00659=1144.767,139.385,-57.472,-178.805,6.892,148.927
C00660=1144.771,139.136,-57.451,-178.808,6.890,148.927
C00661=1144.776,138.886,-57.432,-178.811,6.888,148.928
C00662=1144.781,138.637,-57.411,-178.814,6.887,148.928
C00663=1144.785,138.388,-57.390,-178.816,6.885,148.929
C00664=1144.790,138.139,-57.370,-178.819,6.883,148.929
C00665=1144.794,137.890,-57.350,-178.821,6.881,148.929
C00666=1144.800,137.640,-57.329,-178.825,6.879,148.930
C00667=1144.804,137.391,-57.309,-178.827,6.877,148.930
C00668=1144.809,137.142,-57.289,-178.830,6.875,148.930
C00669=1144.814,136.893,-57.268,-178.833,6.873,148.931
C00670=1144.818,136.644,-57.247,-178.836,6.872,148.931
C00671=1144.823,136.395,-57.228,-178.838,6.870,148.932
C00672=1144.828,136.146,-57.208,-178.841,6.868,148.932
C00673=1144.833,135.897,-57.187,-178.844,6.867,148.932
C00674=1144.838,135.647,-57.167,-178.847,6.864,148.933
C00675=1144.842,135.398,-57.147,-178.850,6.862,148.933
C00676=1144.847,135.150,-57.126,-178.852,6.861,148.933
C00677=1144.852,134.900,-57.106,-178.855,6.859,148.934
C00678=1144.857,134.651,-57.086,-178.858,6.857,148.934
C00679=1144.861,134.402,-57.065,-178.861,6.856,148.935
C00680=1144.867,134.153,-57.046,-178.863,6.854,148.935
C00681=1144.871,133.904,-57.025,-178.866,6.852,148.935
C00682=1144.875,133.655,-57.005,-178.869,6.850,148.936
C00683=1144.881,133.405,-56.985,-178.872,6.848,148.936
C00684=1144.885,133.156,-56.964,-178.875,6.846,148.937
C00685=1144.890,132.907,-56.945,-178.877,6.845,148.937
C00686=1144.894,132.658,-56.924,-178.880,6.843,148.937
C00687=1144.900,132.409,-56.905,-178.883,6.841,148.938
C00688=1144.904,132.160,-56.885,-178.886,6.839,148.938
C00689=1144.910,131.891,-56.863,-178.889,6.837,148.939
C00690=1144.915,131.623,-56.841,-178.892,6.835,148.939
C00691=1144.920,131.354,-56.820,-178.894,6.833,148.939
C00692=1144.925,131.085,-56.799,-178.898,6.831,148.940
C00693=1144.930,130.836,-56.778,-178.900,6.829,148.940
C00694=1144.934,130.587,-56.759,-178.903,6.828,148.941
C00695=1144.939,130.338,-56.739,-178.906,6.826,148.941
C00696=1144.944,130.089,-56.719,-178.909,6.824,148.941
C00697=1144.949,129.839,-56.699,-178.911,6.822,148.942
C00698=1144.953,129.590,-56.679,-178.914,6.821,148.942
C00699=1144.959,129.342,-56.660,-178.917,6.819,148.943
C00700=1144.963,129.093,-56.639,-178.920,6.818,148.943
C00701=1144.968,128.843,-56.619,-178.923,6.816,148.944
C00702=1144.973,128.593,-56.599,-178.925,6.814,148.944
C00703=1144.978,128.345,-56.579,-178.928,6.813,148.944
C00704=1144.983,128.095,-56.560,-178.931,6.811,148.945
C00705=1144.987,127.846,-56.539,-178.934,6.808,148.945
C00706=1144.992,127.597,-56.520,-178.937,6.807,148.945
C00707=1144.997,127.348,-56.501,-178.940,6.805,148.946
C00708=1145.002,127.099,-56.481,-178.942,6.803,148.946
C00709=1145.006,126.850,-56.461,-178.945,6.802,148.947
C00710=1145.011,126.600,-56.441,-178.948,6.800,148.947
C00711=1145.016,126.351,-56.422,-178.950,6.798,148.947
C00712=1145.021,126.102,-56.402,-178.953,6.797,148.948
C00713=1145.025,125.853,-56.382,-178.956,6.795,148.948
C00714=1145.031,125.604,-56.363,-178.959,6.793,148.949
C00715=1145.035,125.354,-56.343,-178.961,6.791,148.949
C00716=1145.040,125.105,-56.323,-178.964,6.790,148.949
C00717=1145.045,124.856,-56.303,-178.967,6.788,148.950
C00718=1145.050,124.607,-56.284,-178.969,6.786,148.950
C00719=1145.054,124.358,-56.265,-178.972,6.785,148.951
C00720=1145.059,124.108,-56.245,-178.975,6.783,148.951
C00721=1145.064,123.860,-56.225,-178.978,6.781,148.951
C00722=1145.068,123.610,-56.205,-178.980,6.780,148.952
C00723=1145.073,123.361,-56.186,-178.983,6.778,148.952
C00724=1145.078,123.112,-56.166,-178.986,6.776,148.953
C00725=1145.083,122.862,-56.147,-178.989,6.774,148.953
C00726=1145.088,122.614,-56.128,-178.992,6.772,148.953
C00727=1145.093,122.364,-56.108,-178.995,6.770,148.954
C00728=1145.097,122.115,-56.089,-178.998,6.769,148.954
C00729=1145.103,121.866,-56.069,-179.000,6.767,148.955
C00730=1145.107,121.616,-56.050,-179.003,6.765,148.955
C00731=1145.111,121.368,-56.030,-179.006,6.764,148.956
C00732=1145.116,121.119,-56.011,-179.009,6.762,148.956
C00733=1145.121,120.869,-55.991,-179.011,6.760,148.956
C00734=1145.127,120.620,-55.972,-179.014,6.759,148.957
C00735=1145.131,120.371,-55.953,-179.017,6.757,148.957
C00736=1145.135,120.121,-55.933,-179.020,6.755,148.958
C00737=1145.141,119.873,-55.914,-179.022,6.754,148.958
C00738=1145.145,119.623,-55.894,-179.025,6.752,148.958
C00739=1145.150,119.374,-55.875,-179.028,6.750,148.959
C00740=1145.155,119.125,-55.856,-179.030,6.749,148.959
C00741=1145.160,118.875,-55.837,-179.033,6.747,148.960
C00742=1145.165,118.626,-55.817,-179.036,6.745,148.960
C00743=1145.169,118.377,-55.798,-179.039,6.744,148.961
C00744=1145.174,118.128,-55.779,-179.042,6.742,148.961
C00745=1145.179,117.878,-55.759,-179.045,6.740,148.962
C00746=1145.184,117.630,-55.741,-179.047,6.739,148.962
C00747=1145.189,117.380,-55.721,-179.050,6.737,148.962
C00748=1145.194,117.131,-55.702,-179.053,6.735,148.963
C00749=1145.198,116.882,-55.683,-179.055,6.734,148.963
C00750=1145.204,116.632,-55.664,-179.058,6.732,148.964
C00751=1145.208,116.383,-55.644,-179.061,6.730,148.964
C00752=1145.213,116.134,-55.626,-179.064,6.729,148.964
C00753=1145.218,115.885,-55.606,-179.066,6.727,148.965
C00754=1145.223,115.636,-55.587,-179.070,6.726,148.965
C00755=1145.227,115.386,-55.568,-179.072,6.725,148.966
C00756=1145.233,115.137,-55.549,-179.074,6.723,148.966
C00757=1145.237,114.888,-55.530,-179.077,6.721,148.967
C00758=1145.242,114.639,-55.511,-179.080,6.720,148.967
C00759=1145.247,114.389,-55.492,-179.083,6.718,148.967
C00760=1145.252,114.140,-55.473,-179.085,6.716,148.968
C00761=1145.256,113.891,-55.454,-179.088,6.715,148.968
C00762=1145.261,113.642,-55.435,-179.091,6.713,148.969
C00763=1145.267,113.393,-55.416,-179.093,6.711,148.969
C00764=1145.271,113.143,-55.397,-179.097,6.710,148.970
C00765=1145.276,112.894,-55.378,-179.099,6.708,148.970
C00766=1145.280,112.645,-55.360,-179.102,6.706,148.971
C00767=1145.286,112.396,-55.340,-179.105,6.705,148.971
C00768=1145.290,112.146,-55.321,-179.108,6.703,148.971
C00769=1145.295,111.897,-55.303,-179.110,6.701,148.972
C00770=1145.301,111.648,-55.283,-179.113,6.700,148.972
C00771=1145.305,111.399,-55.264,-179.116,6.698,148.973
C00772=1145.310,111.149,-55.246,-179.118,6.696,148.973
C00773=1145.314,110.900,-55.227,-179.122,6.695,148.974
C00774=1145.319,110.651,-55.209,-179.124,6.693,148.974
C00775=1145.325,110.402,-55.189,-179.127,6.692,148.974
C00776=1145.329,110.152,-55.171,-179.129,6.691,148.975
C00777=1145.334,109.903,-55.152,-179.132,6.689,148.975
C00778=1145.338,109.654,-55.133,-179.135,6.687,148.976
C00779=1145.344,109.405,-55.114,-179.137,6.686,148.976
C00780=1145.348,109.156,-55.095,-179.141,6.684,148.977
C00781=1145.354,108.906,-55.076,-179.143,6.683,148.977
C00782=1145.358,108.657,-55.058,-179.146,6.681,148.977
C00783=1145.363,108.408,-55.040,-179.149,6.679,148.978
C00784=1145.368,108.159,-55.020,-179.152,6.678,148.978
C00785=1145.373,107.909,-55.002,-179.154,6.676,148.979
C00786=1145.377,107.659,-54.984,-179.157,6.674,148.979
C00787=1145.382,107.411,-54.965,-179.160,6.672,148.980
C00788=1145.387,107.161,-54.947,-179.163,6.671,148.980
C00789=1145.392,106.912,-54.927,-179.165,6.670,148.981
C00790=1145.397,106.663,-54.909,-179.168,6.669,148.981
C00791=1145.402,106.414,-54.890,-179.171,6.667,148.981
C00792=1145.407,106.164,-54.871,-179.173,6.665,148.982
C00793=1145.412,105.896,-54.852,-179.176,6.664,148.982
C00794=1145.417,105.627,-54.832,-179.179,6.662,148.983
C00795=1145.422,105.359,-54.812,-179.182,6.661,148.983
C00796=1145.427,105.091,-54.792,-179.185,6.658,148.984
C00797=1145.432,104.841,-54.773,-179.188,6.658,148.984
C00798=1145.437,104.592,-54.755,-179.191,6.656,148.985
C00799=1145.442,104.343,-54.737,-179.193,6.654,148.985
C00800=1145.448,104.094,-54.718,-179.196,6.652,148.986
C00801=1145.452,103.844,-54.700,-179.199,6.651,148.986
C00802=1145.456,103.595,-54.681,-179.202,6.649,148.986
C00803=1145.461,103.346,-54.663,-179.205,6.648,148.987
C00804=1145.466,103.096,-54.644,-179.207,6.646,148.987
C00805=1145.471,102.847,-54.626,-179.210,6.644,148.988
C00806=1145.476,102.598,-54.608,-179.212,6.644,148.988
C00807=1145.481,102.349,-54.590,-179.215,6.642,148.989
C00808=1145.487,102.100,-54.571,-179.218,6.640,148.989
C00809=1145.491,101.850,-54.553,-179.221,6.639,148.990
C00810=1145.495,101.601,-54.534,-179.224,6.637,148.990
C00811=1145.500,101.352,-54.516,-179.226,6.635,148.991
C00812=1145.505,101.103,-54.498,-179.229,6.634,148.991
C00813=1145.510,100.853,-54.479,-179.232,6.632,148.991
C00814=1145.515,100.603,-54.461,-179.234,6.631,148.992
C00815=1145.520,100.354,-54.443,-179.237,6.630,148.992
C00816=1145.525,100.105,-54.425,-179.240,6.628,148.993
C00817=1145.530,99.857,-54.406,-179.243,6.627,148.993
C00818=1145.534,99.607,-54.388,-179.246,6.625,148.994
C00819=1145.539,99.358,-54.370,-179.248,6.623,148.994
C00820=1145.545,99.108,-54.351,-179.251,6.622,148.995
C00821=1145.549,98.859,-54.334,-179.254,6.621,148.995
C00822=1145.554,98.610,-54.316,-179.256,6.619,148.996
C00823=1145.559,98.361,-54.298,-179.259,6.618,148.996
C00824=1145.564,98.111,-54.279,-179.262,6.616,148.996
C00825=1145.568,97.861,-54.261,-179.265,6.615,148.997
C00826=1145.573,97.612,-54.243,-179.268,6.613,148.997
C00827=1145.578,97.363,-54.225,-179.270,6.612,148.998
C00828=1145.583,97.114,-54.207,-179.273,6.610,148.998
C00829=1145.588,96.865,-54.189,-179.275,6.609,148.999
C00830=1145.592,96.615,-54.171,-179.278,6.607,148.999
C00831=1145.597,96.366,-54.153,-179.281,6.606,149.000
C00832=1145.603,96.116,-54.134,-179.284,6.604,149.000
C00833=1145.608,95.867,-54.116,-179.286,6.603,149.001
C00834=1145.613,95.618,-54.098,-179.289,6.601,149.001
C00835=1145.618,95.369,-54.080,-179.292,6.600,149.002
C00836=1145.623,95.120,-54.062,-179.295,6.598,149.002
C00837=1145.628,94.870,-54.045,-179.298,6.597,149.003
C00838=1145.633,94.621,-54.027,-179.300,6.596,149.003
C00839=1145.638,94.371,-54.009,-179.302,6.594,149.003
C00840=1145.642,94.121,-53.991,-179.306,6.593,149.004
C00841=1145.647,93.872,-53.973,-179.308,6.591,149.004
C00842=1145.652,93.623,-53.955,-179.311,6.590,149.005
C00843=1145.656,93.374,-53.938,-179.314,6.588,149.005
C00844=1145.661,93.125,-53.920,-179.316,6.587,149.006
C00845=1145.666,92.875,-53.902,-179.319,6.586,149.006
C00846=1145.671,92.626,-53.884,-179.322,6.584,149.007
C00847=1145.676,92.377,-53.866,-179.325,6.582,149.007
C00848=1145.681,92.128,-53.848,-179.327,6.581,149.008
C00849=1145.686,91.879,-53.830,-179.330,6.580,149.008
C00850=1145.691,91.629,-53.813,-179.333,6.579,149.009
C00851=1145.696,91.380,-53.795,-179.336,6.577,149.009
C00852=1145.701,91.130,-53.777,-179.338,6.575,149.009
C00853=1145.706,90.881,-53.759,-179.340,6.574,149.010
C00854=1145.711,90.631,-53.742,-179.344,6.573,149.011
C00855=1145.715,90.383,-53.725,-179.346,6.571,149.011
C00856=1145.720,90.133,-53.707,-179.349,6.570,149.011
C00857=1145.725,89.884,-53.689,-179.352,6.568,149.012
C00858=1145.730,89.634,-53.671,-179.354,6.567,149.012
C00859=1145.735,89.385,-53.653,-179.357,6.566,149.013
C00860=1145.740,89.136,-53.636,-179.360,6.564,149.013
C00861=1145.745,88.886,-53.618,-179.363,6.562,149.014
C00862=1145.749,88.637,-53.601,-179.365,6.561,149.014
C00863=1145.755,88.388,-53.583,-179.368,6.560,149.015
C00864=1145.760,88.139,-53.565,-179.371,6.559,149.015
C00865=1145.764,87.889,-53.547,-179.374,6.557,149.016
C00866=1145.770,87.640,-53.530,-179.376,6.555,149.016
C00867=1145.774,87.391,-53.513,-179.379,6.555,149.017
C00868=1145.779,87.141,-53.496,-179.382,6.553,149.017
C00869=1145.784,86.892,-53.478,-179.384,6.551,149.018
C00870=1145.789,86.642,-53.460,-179.387,6.550,149.018
C00871=1145.793,86.393,-53.443,-179.390,6.549,149.019
C00872=1145.798,86.144,-53.425,-179.392,6.548,149.019
C00873=1145.803,85.894,-53.408,-179.395,6.546,149.019
C00874=1145.808,85.645,-53.390,-179.398,6.544,149.020
C00875=1145.813,85.395,-53.373,-179.401,6.544,149.021
C00876=1145.818,85.147,-53.355,-179.403,6.542,149.021
C00877=1145.824,84.897,-53.338,-179.406,6.540,149.021
C00878=1145.828,84.648,-53.320,-179.409,6.539,149.022
C00879=1145.833,84.398,-53.304,-179.411,6.538,149.022
C00880=1145.838,84.149,-53.286,-179.414,6.537,149.023
C00881=1145.843,83.899,-53.268,-179.417,6.535,149.023
C00882=1145.848,83.650,-53.252,-179.420,6.533,149.024
C00883=1145.853,83.401,-53.234,-179.422,6.533,149.024
C00884=1145.858,83.151,-53.216,-179.425,6.531,149.025
C00885=1145.862,82.902,-53.199,-179.428,6.529,149.025
C00886=1145.868,82.653,-53.182,-179.430,6.528,149.026
C00887=1145.873,82.403,-53.165,-179.433,6.527,149.026
C00888=1145.877,82.154,-53.147,-179.436,6.525,149.027
C00889=1145.882,81.905,-53.130,-179.439,6.524,149.027
C00890=1145.887,81.655,-53.114,-179.441,6.523,149.028
C00891=1145.892,81.406,-53.096,-179.444,6.522,149.028
C00892=1145.897,81.156,-53.078,-179.447,6.520,149.029
C00893=1145.902,80.907,-53.062,-179.449,6.518,149.029
C00894=1145.907,80.658,-53.044,-179.452,6.518,149.030
C00895=1145.911,80.409,-53.027,-179.455,6.516,149.030
C00896=1145.917,80.159,-53.010,-179.458,6.514,149.031
C00897=1145.923,79.891,-52.992,-179.461,6.513,149.031
C00898=1145.927,79.623,-52.973,-179.463,6.512,149.032
C00899=1145.932,79.354,-52.954,-179.466,6.511,149.032
C00900=1145.938,79.086,-52.936,-179.469,6.509,149.033
C00901=1145.943,78.836,-52.919,-179.472,6.508,149.033
C00902=1145.948,78.587,-52.902,-179.474,6.506,149.034
C00903=1145.953,78.337,-52.885,-179.477,6.506,149.034
C00904=1145.958,78.089,-52.868,-179.480,6.504,149.035
C00905=1145.963,77.839,-52.851,-179.482,6.502,149.035
C00906=1145.968,77.589,-52.834,-179.485,6.502,149.036
C00907=1145.972,77.340,-52.817,-179.488,6.500,149.036
C00908=1145.977,77.090,-52.800,-179.491,6.498,149.037
C00909=1145.982,76.842,-52.783,-179.493,6.497,149.037
C00910=1145.987,76.592,-52.766,-179.496,6.496,149.038
C00911=1145.992,76.343,-52.749,-179.499,6.495,149.038
C00912=1145.997,76.093,-52.732,-179.501,6.493,149.039
C00913=1146.002,75.844,-52.715,-179.504,6.492,149.039
C00914=1146.007,75.594,-52.698,-179.507,6.491,149.040
C00915=1146.012,75.345,-52.681,-179.510,6.489,149.040
C00916=1146.016,75.095,-52.665,-179.512,6.488,149.041
C00917=1146.022,74.846,-52.648,-179.515,6.487,149.041
C00918=1146.027,74.597,-52.631,-179.518,6.485,149.042
C00919=1146.032,74.347,-52.613,-179.520,6.484,149.042
C00920=1146.037,74.099,-52.597,-179.523,6.483,149.043
C00921=1146.042,73.849,-52.580,-179.526,6.481,149.043
C00922=1146.046,73.599,-52.563,-179.528,6.481,149.044
C00923=1146.051,73.351,-52.547,-179.531,6.479,149.044
C00924=1146.057,73.101,-52.529,-179.534,6.478,149.045
C00925=1146.061,72.851,-52.513,-179.536,6.477,149.045
C00926=1146.066,72.602,-52.496,-179.539,6.475,149.046
C00927=1146.071,72.353,-52.479,-179.542,6.474,149.046
C00928=1146.076,72.103,-52.462,-179.544,6.473,149.047
C00929=1146.081,71.853,-52.446,-179.547,6.471,149.047
C00930=1146.087,71.604,-52.430,-179.550,6.470,149.048
C00931=1146.091,71.355,-52.413,-179.552,6.469,149.048
C00932=1146.096,71.105,-52.396,-179.555,6.467,149.049
C00933=1146.101,70.856,-52.379,-179.558,6.467,149.049
C00934=1146.106,70.607,-52.363,-179.560,6.465,149.050
C00935=1146.111,70.358,-52.346,-179.563,6.464,149.050
C00936=1146.116,70.108,-52.329,-179.565,6.463,149.051
C00937=1146.121,69.858,-52.312,-179.569,6.461,149.051
C00938=1146.126,69.610,-52.296,-179.571,6.460,149.052
C00939=1146.131,69.359,-52.280,-179.573,6.459,149.052
C00940=1146.136,69.110,-52.263,-179.577,6.458,149.053
C00941=1146.141,68.861,-52.247,-179.579,6.456,149.053
C00942=1146.145,68.612,-52.230,-179.582,6.455,149.054
C00943=1146.151,68.362,-52.213,-179.585,6.454,149.054
C00944=1146.156,68.113,-52.196,-179.587,6.453,149.055
C00945=1146.160,67.863,-52.180,-179.590,6.451,149.055
C00946=1146.165,67.614,-52.164,-179.593,6.450,149.056
C00947=1146.171,67.364,-52.147,-179.595,6.449,149.056
C00948=1146.176,67.115,-52.131,-179.598,6.448,149.057
C00949=1146.180,66.865,-52.115,-179.600,6.447,149.057
C00950=1146.185,66.616,-52.098,-179.603,6.445,149.058
C00951=1146.190,66.367,-52.082,-179.606,6.444,149.058
C00952=1146.195,66.117,-52.064,-179.609,6.443,149.059
C00953=1146.201,65.868,-52.049,-179.611,6.442,149.059
C00954=1146.205,65.618,-52.032,-179.614,6.440,149.060
C00955=1146.210,65.370,-52.016,-179.617,6.439,149.060
C00956=1146.215,65.120,-52.000,-179.619,6.438,149.061
C00957=1146.219,64.870,-51.983,-179.622,6.437,149.061
C00958=1146.225,64.621,-51.966,-179.625,6.436,149.062
C00959=1146.230,64.371,-51.950,-179.628,6.434,149.062
C00960=1146.235,64.122,-51.934,-179.630,6.433,149.063
C00961=1146.240,63.873,-51.917,-179.633,6.432,149.063
C00962=1146.245,63.623,-51.902,-179.635,6.431,149.064
C00963=1146.249,63.374,-51.885,-179.638,6.429,149.064
C00964=1146.255,63.124,-51.869,-179.640,6.429,149.065
C00965=1146.259,62.875,-51.853,-179.643,6.427,149.065
C00966=1146.264,62.626,-51.837,-179.646,6.426,149.066
C00967=1146.270,62.376,-51.820,-179.649,6.425,149.066
C00968=1146.275,62.127,-51.804,-179.651,6.423,149.067
C00969=1146.280,61.877,-51.788,-179.654,6.423,149.067
C00970=1146.285,61.628,-51.771,-179.657,6.421,149.068
C00971=1146.290,61.378,-51.755,-179.659,6.420,149.068
C00972=1146.295,61.129,-51.739,-179.662,6.419,149.069
C00973=1146.300,60.879,-51.723,-179.665,6.417,149.070
C00974=1146.305,60.630,-51.707,-179.667,6.417,149.070
C00975=1146.309,60.380,-51.691,-179.670,6.415,149.070
C00976=1146.315,60.131,-51.675,-179.672,6.415,149.071
C00977=1146.320,59.882,-51.659,-179.675,6.413,149.072
C00978=1146.324,59.632,-51.642,-179.677,6.412,149.072
C00979=1146.330,59.383,-51.627,-179.681,6.411,149.073
C00980=1146.334,59.134,-51.610,-179.683,6.409,149.073
C00981=1146.340,58.884,-51.595,-179.685,6.408,149.074
C00982=1146.344,58.635,-51.578,-179.689,6.407,149.074
C00983=1146.349,58.385,-51.562,-179.691,6.406,149.075
C00984=1146.355,58.136,-51.547,-179.694,6.404,149.075
C00985=1146.359,57.886,-51.530,-179.696,6.404,149.076
C00986=1146.365,57.637,-51.514,-179.699,6.402,149.076
C00987=1146.369,57.387,-51.498,-179.701,6.401,149.077
C00988=1146.375,57.138,-51.482,-179.704,6.400,149.077
C00989=1146.379,56.888,-51.466,-179.707,6.399,149.078
C00990=1146.384,56.639,-51.450,-179.710,6.398,149.078
C00991=1146.390,56.390,-51.434,-179.713,6.396,149.079
C00992=1146.394,56.140,-51.419,-179.715,6.396,149.079
C00993=1146.399,55.891,-51.403,-179.718,6.394,149.080
C00994=1146.404,55.642,-51.387,-179.720,6.393,149.080
C00995=1146.409,55.392,-51.371,-179.723,6.392,149.081
C00996=1146.414,55.143,-51.355,-179.725,6.391,149.081
C00997=1146.420,54.893,-51.339,-179.728,6.390,149.082
C00998=1146.424,54.643,-51.323,-179.730,6.389,149.082
C00999=1146.430,54.394,-51.308,-179.734,6.388,149.083
C01000=1146.434,54.144,-51.291,-179.736,6.387,149.083
C01001=1146.440,53.876,-51.274,-179.739,6.385,149.084
C01002=1146.445,53.607,-51.258,-179.742,6.384,149.085
C01003=1146.451,53.339,-51.241,-179.745,6.382,149.085
C01004=1146.456,53.070,-51.224,-179.747,6.382,149.086
C01005=1146.461,52.821,-51.208,-179.750,6.380,149.086
C01006=1146.466,52.571,-51.192,-179.753,6.379,149.087
C01007=1146.471,52.322,-51.176,-179.755,6.378,149.087
C01008=1146.476,52.072,-51.160,-179.758,6.377,149.088
C01009=1146.481,51.823,-51.145,-179.761,6.376,149.088
C01010=1146.486,51.573,-51.130,-179.763,6.375,149.089
C01011=1146.491,51.325,-51.114,-179.766,6.374,149.089
C01012=1146.496,51.074,-51.098,-179.768,6.373,149.090
C01013=1146.501,50.825,-51.083,-179.771,6.371,149.091
C01014=1146.506,50.576,-51.067,-179.774,6.371,149.091
C01015=1146.511,50.326,-51.051,-179.776,6.369,149.091
C01016=1146.516,50.076,-51.036,-179.779,6.369,149.092
C01017=1146.521,49.827,-51.021,-179.782,6.367,149.093
C01018=1146.526,49.578,-51.005,-179.784,6.366,149.093
C01019=1146.531,49.328,-50.989,-179.787,6.365,149.094
C01020=1146.536,49.078,-50.973,-179.789,6.364,149.094
C01021=1146.541,48.829,-50.958,-179.793,6.363,149.095
C01022=1146.546,48.580,-50.943,-179.795,6.362,149.095
C01023=1146.551,48.330,-50.927,-179.797,6.360,149.096
C01024=1146.556,48.081,-50.911,-179.800,6.360,149.096
C01025=1146.561,47.832,-50.896,-179.803,6.358,149.097
C01026=1146.566,47.583,-50.880,-179.805,6.358,149.097
C01027=1146.570,47.333,-50.865,-179.808,6.356,149.098
C01028=1146.576,47.083,-50.850,-179.810,6.355,149.098
C01029=1146.582,46.833,-50.834,-179.814,6.354,149.099
C01030=1146.586,46.584,-50.819,-179.816,6.353,149.099
C01031=1146.591,46.334,-50.803,-179.819,6.351,149.100
C01032=1146.596,46.085,-50.788,-179.821,6.351,149.101
C01033=1146.601,45.836,-50.773,-179.823,6.350,149.101
C01034=1146.606,45.586,-50.757,-179.827,6.349,149.102
C01035=1146.612,45.337,-50.741,-179.829,6.348,149.102
C01036=1146.616,45.087,-50.726,-179.831,6.346,149.103
C01037=1146.621,44.838,-50.711,-179.834,6.346,149.103
C01038=1146.626,44.589,-50.696,-179.837,6.344,149.104
C01039=1146.631,44.339,-50.680,-179.840,6.344,149.104
C01040=1146.637,44.089,-50.665,-179.842,6.342,149.105
C01041=1146.642,43.840,-50.650,-179.844,6.341,149.105
C01042=1146.646,43.590,-50.634,-179.848,6.340,149.106
C01043=1146.651,43.341,-50.619,-179.850,6.339,149.106
C01044=1146.656,43.092,-50.604,-179.852,6.338,149.107
C01045=1146.661,42.842,-50.589,-179.855,6.337,149.107
C01046=1146.667,42.592,-50.574,-179.857,6.336,149.108
C01047=1146.672,42.343,-50.558,-179.861,6.335,149.109
C01048=1146.677,42.094,-50.543,-179.863,6.334,149.109
C01049=1146.682,41.844,-50.527,-179.866,6.332,149.110
C01050=1146.686,41.595,-50.512,-179.868,6.332,149.110
C01051=1146.692,41.345,-50.497,-179.871,6.330,149.111
C01052=1146.697,41.096,-50.482,-179.874,6.330,149.111
C01053=1146.702,40.846,-50.467,-179.876,6.329,149.112
C01054=1146.707,40.597,-50.452,-179.879,6.327,149.112
C01055=1146.712,40.347,-50.437,-179.881,6.327,149.113
C01056=1146.717,40.098,-50.422,-179.884,6.325,149.113
C01057=1146.722,39.849,-50.406,-179.887,6.325,149.114
C01058=1146.727,39.598,-50.392,-179.889,6.323,149.114
C01059=1146.732,39.349,-50.376,-179.891,6.322,149.115
C01060=1146.737,39.100,-50.361,-179.894,6.322,149.116
C01061=1146.742,38.850,-50.346,-179.897,6.320,149.116
C01062=1146.747,38.601,-50.331,-179.900,6.320,149.117
C01063=1146.752,38.351,-50.316,-179.902,6.318,149.117
C01064=1146.757,38.101,-50.301,-179.904,6.317,149.118
C01065=1146.762,37.852,-50.286,-179.907,6.317,149.118
C01066=1146.767,37.603,-50.271,-179.910,6.315,149.119
C01067=1146.772,37.353,-50.256,-179.913,6.315,149.119
C01068=1146.778,37.104,-50.241,-179.915,6.313,149.120
C01069=1146.783,36.854,-50.227,-179.917,6.312,149.120
C01070=1146.787,36.605,-50.212,-179.920,6.312,149.121
C01071=1146.793,36.356,-50.196,-179.923,6.310,149.121
C01072=1146.798,36.106,-50.182,-179.925,6.310,149.122
C01073=1146.803,35.857,-50.166,-179.928,6.308,149.123
C01074=1146.808,35.607,-50.152,-179.930,6.307,149.123
C01075=1146.813,35.358,-50.137,-179.933,6.307,149.124
C01076=1146.818,35.108,-50.122,-179.936,6.305,149.124
C01077=1146.823,34.859,-50.107,-179.938,6.305,149.125
C01078=1146.828,34.609,-50.093,-179.941,6.303,149.125
C01079=1146.833,34.360,-50.077,-179.943,6.302,149.126
C01080=1146.838,34.110,-50.063,-179.946,6.302,149.126
C01081=1146.843,33.861,-50.048,-179.949,6.300,149.127
C01082=1146.849,33.611,-50.033,-179.951,6.300,149.127
C01083=1146.853,33.362,-50.018,-179.954,6.298,149.128
C01084=1146.858,33.112,-50.004,-179.957,6.297,149.129
C01085=1146.864,32.862,-49.988,-179.959,6.297,149.129
C01086=1146.869,32.613,-49.974,-179.962,6.295,149.130
C01087=1146.874,32.363,-49.960,-179.964,6.295,149.130
C01088=1146.879,32.114,-49.944,-179.967,6.294,149.131
C01089=1146.884,31.864,-49.930,-179.970,6.292,149.131
C01090=1146.889,31.615,-49.915,-179.972,6.292,149.132
C01091=1146.894,31.365,-49.900,-179.975,6.290,149.132
C01092=1146.899,31.115,-49.886,-179.977,6.290,149.133
C01093=1146.904,30.866,-49.871,-179.980,6.289,149.133
C01094=1146.909,30.616,-49.856,-179.983,6.287,149.134
C01095=1146.914,30.367,-49.842,-179.985,6.287,149.134
C01096=1146.919,30.117,-49.826,-179.987,6.286,149.135
C01097=1146.924,29.867,-49.812,-179.990,6.285,149.136
C01098=1146.929,29.618,-49.798,-179.993,6.284,149.136
C01099=1146.934,29.369,-49.783,-179.995,6.283,149.137
C01100=1146.939,29.120,-49.769,-179.998,6.282,149.137
C01101=1146.945,28.870,-49.754,179.999,6.281,149.138
C01102=1146.950,28.621,-49.739,179.997,6.280,149.138
C01103=1146.955,28.371,-49.725,179.994,6.279,149.139
C01104=1146.960,28.121,-49.711,179.992,6.278,149.139
C01105=1146.965,27.852,-49.695,179.989,6.277,149.140
C01106=1146.971,27.583,-49.679,179.986,6.276,149.141
C01107=1146.976,27.314,-49.664,179.983,6.275,149.141
C01108=1146.981,27.045,-49.648,179.981,6.274,149.142
C01109=1146.987,26.796,-49.634,179.978,6.273,149.142
C01110=1146.991,26.547,-49.619,179.976,6.272,149.143
C01111=1146.997,26.297,-49.604,179.973,6.272,149.144
C01112=1147.002,26.047,-49.590,179.970,6.270,149.144
C01113=1147.007,25.798,-49.576,179.968,6.269,149.144
C01114=1147.012,25.548,-49.561,179.965,6.269,149.145
C01115=1147.016,25.299,-49.546,179.963,6.267,149.146
C01116=1147.022,25.050,-49.532,179.960,6.267,149.146
C01117=1147.027,24.800,-49.518,179.958,6.266,149.147
C01118=1147.032,24.550,-49.504,179.955,6.264,149.147
C01119=1147.037,24.301,-49.489,179.952,6.264,149.148
C01120=1147.042,24.051,-49.475,179.950,6.263,149.148
C01121=1147.048,23.801,-49.460,179.947,6.262,149.149
C01122=1147.053,23.552,-49.446,179.945,6.261,149.149
C01123=1147.058,23.302,-49.432,179.942,6.260,149.150
C01124=1147.063,23.053,-49.417,179.940,6.259,149.151
C01125=1147.068,22.803,-49.403,179.937,6.258,149.151
C01126=1147.073,22.554,-49.389,179.935,6.257,149.152
C01127=1147.078,22.305,-49.375,179.932,6.257,149.152
C01128=1147.083,22.055,-49.360,179.929,6.255,149.153
C01129=1147.088,21.805,-49.346,179.927,6.254,149.153
C01130=1147.093,21.555,-49.332,179.924,6.254,149.154
C01131=1147.098,21.306,-49.318,179.922,6.252,149.154
C01132=1147.104,21.057,-49.304,179.919,6.252,149.155
C01133=1147.109,20.807,-49.289,179.917,6.251,149.156
C01134=1147.113,20.557,-49.275,179.915,6.250,149.156
C01135=1147.118,20.308,-49.261,179.911,6.249,149.157
C01136=1147.124,20.059,-49.247,179.909,6.248,149.157
C01137=1147.129,19.809,-49.233,179.907,6.248,149.158
C01138=1147.134,19.559,-49.218,179.904,6.246,149.158
C01139=1147.139,19.309,-49.204,179.901,6.246,149.159
C01140=1147.144,19.060,-49.190,179.899,6.245,149.159
C01141=1147.149,18.811,-49.176,179.897,6.244,149.160
C01142=1147.154,18.561,-49.162,179.894,6.243,149.161
C01143=1147.159,18.311,-49.149,179.891,6.242,149.161
C01144=1147.164,18.062,-49.135,179.889,6.242,149.162
C01145=1147.169,17.812,-49.120,179.886,6.240,149.162
C01146=1147.174,17.563,-49.106,179.883,6.239,149.163
C01147=1147.180,17.314,-49.092,179.881,6.239,149.163
C01148=1147.185,17.064,-49.078,179.879,6.238,149.164
C01149=1147.190,16.814,-49.064,179.876,6.237,149.164
C01150=1147.195,16.564,-49.049,179.874,6.236,149.165
C01151=1147.201,16.315,-49.036,179.871,6.235,149.166
C01152=1147.205,16.065,-49.023,179.869,6.234,149.166
C01153=1147.210,15.816,-49.008,179.865,6.233,149.167
C01154=1147.215,15.567,-48.994,179.863,6.232,149.167
C01155=1147.220,15.317,-48.980,179.861,6.232,149.168
C01156=1147.225,15.067,-48.966,179.858,6.230,149.168
C01157=1147.231,14.818,-48.953,179.856,6.230,149.169
C01158=1147.236,14.568,-48.938,179.853,6.229,149.169
C01159=1147.240,14.319,-48.925,179.851,6.228,149.170
C01160=1147.246,14.070,-48.911,179.848,6.227,149.171
C01161=1147.251,13.819,-48.897,179.845,6.226,149.171
C01162=1147.256,13.569,-48.883,179.843,6.226,149.172
C01163=1147.262,13.320,-48.869,179.841,6.225,149.172
C01164=1147.266,13.071,-48.855,179.838,6.223,149.173
C01165=1147.271,12.821,-48.842,179.835,6.223,149.173
C01166=1147.277,12.572,-48.828,179.833,6.222,149.174
C01167=1147.282,12.322,-48.814,179.830,6.222,149.175
C01168=1147.287,12.072,-48.800,179.828,6.220,149.175
C01169=1147.292,11.823,-48.787,179.825,6.220,149.176
C01170=1147.297,11.573,-48.772,179.823,6.219,149.176
C01171=1147.302,11.324,-48.759,179.821,6.218,149.177
C01172=1147.307,11.074,-48.745,179.818,6.217,149.177
C01173=1147.312,10.825,-48.731,179.815,6.216,149.178
C01174=1147.317,10.575,-48.718,179.813,6.215,149.178
C01175=1147.322,10.325,-48.704,179.810,6.215,149.179
C01176=1147.328,10.076,-48.690,179.808,6.214,149.180
C01177=1147.333,9.826,-48.677,179.805,6.213,149.180
C01178=1147.338,9.577,-48.663,179.802,6.212,149.181
C01179=1147.343,9.327,-48.649,179.800,6.211,149.181
C01180=1147.348,9.077,-48.636,179.798,6.210,149.182
C01181=1147.353,8.828,-48.622,179.795,6.210,149.182
C01182=1147.358,8.578,-48.608,179.793,6.208,149.183
C01183=1147.363,8.329,-48.595,179.790,6.208,149.183
C01184=1147.368,8.079,-48.581,179.788,6.207,149.184
C01185=1147.374,7.830,-48.568,179.785,6.207,149.185
C01186=1147.379,7.580,-48.555,179.782,6.205,149.185
C01187=1147.383,7.330,-48.540,179.780,6.205,149.186
C01188=1147.389,7.081,-48.527,179.777,6.204,149.186
C01189=1147.394,6.831,-48.513,179.775,6.203,149.187
C01190=1147.399,6.582,-48.500,179.773,6.203,149.187
C01191=1147.404,6.332,-48.486,179.770,6.201,149.188
C01192=1147.410,6.083,-48.473,179.767,6.200,149.189
C01193=1147.414,5.833,-48.459,179.765,6.200,149.189
C01194=1147.420,5.584,-48.446,179.762,6.199,149.190
C01195=1147.425,5.334,-48.432,179.760,6.198,149.190
C01196=1147.430,5.084,-48.419,179.757,6.197,149.191
C01197=1147.435,4.835,-48.405,179.755,6.196,149.191
C01198=1147.440,4.585,-48.392,179.753,6.196,149.192
C01199=1147.445,4.335,-48.379,179.750,6.195,149.192
C01200=1147.451,4.086,-48.365,179.748,6.194,149.193
C01201=1147.456,3.836,-48.352,179.745,6.193,149.194
C01202=1147.461,3.587,-48.338,179.742,6.192,149.194
C01203=1147.466,3.337,-48.325,179.740,6.192,149.195
C01204=1147.471,3.088,-48.312,179.738,6.191,149.195
C01205=1147.476,2.838,-48.298,179.735,6.191,149.196
C01206=1147.481,2.589,-48.285,179.733,6.190,149.196
C01207=1147.486,2.339,-48.271,179.730,6.188,149.197
C01208=1147.491,2.090,-48.258,179.727,6.188,149.197
C01209=1147.497,1.819,-48.244,179.725,6.187,149.198
C01210=1147.503,1.551,-48.230,179.722,6.186,149.199
C01211=1147.508,1.281,-48.216,179.719,6.185,149.199
C01212=1147.513,1.012,-48.201,179.717,6.184,149.200
C01213=1147.519,0.762,-48.188,179.714,6.184,149.200
C01214=1147.524,0.512,-48.175,179.712,6.182,149.201
C01215=1147.529,0.263,-48.161,179.709,6.182,149.202
C01216=1147.534,0.013,-48.148,179.707,6.181,149.202
C01217=1147.540,-0.237,-48.135,179.704,6.181,149.203
C01218=1147.545,-0.485,-48.121,179.702,6.180,149.203
C01219=1147.550,-0.736,-48.108,179.699,6.179,149.204
C01220=1147.555,-0.985,-48.095,179.697,6.179,149.204
C01221=1147.559,-1.235,-48.082,179.694,6.177,149.205
C01222=1147.565,-1.485,-48.069,179.692,6.177,149.206
C01223=1147.570,-1.733,-48.056,179.690,6.176,149.206
C01224=1147.575,-1.984,-48.042,179.687,6.175,149.207
C01225=1147.580,-2.233,-48.029,179.685,6.175,149.207
C01226=1147.586,-2.483,-48.016,179.682,6.174,149.208
C01227=1147.591,-2.733,-48.003,179.679,6.172,149.208
C01228=1147.596,-2.981,-47.990,179.677,6.172,149.209
C01229=1147.601,-3.232,-47.976,179.674,6.171,149.209
C01230=1147.606,-3.481,-47.964,179.672,6.170,149.210
C01231=1147.611,-3.731,-47.950,179.670,6.170,149.211
C01232=1147.616,-3.981,-47.938,179.667,6.169,149.211
C01233=1147.622,-4.230,-47.925,179.665,6.169,149.212
C01234=1147.627,-4.480,-47.912,179.662,6.167,149.212
C01235=1147.632,-4.729,-47.898,179.659,6.167,149.213
C01236=1147.637,-4.978,-47.886,179.657,6.166,149.213
C01237=1147.642,-5.229,-47.872,179.654,6.165,149.214
C01238=1147.647,-5.478,-47.859,179.652,6.165,149.215
C01239=1147.652,-5.727,-47.847,179.650,6.164,149.215
C01240=1147.658,-5.978,-47.833,179.647,6.163,149.216
C01241=1147.663,-6.227,-47.821,179.645,6.163,149.216
C01242=1147.668,-6.476,-47.808,179.642,6.161,149.217
C01243=1147.673,-6.727,-47.795,179.640,6.161,149.217
C01244=1147.678,-6.976,-47.782,179.637,6.160,149.218
C01245=1147.683,-7.225,-47.769,179.635,6.159,149.219
C01246=1147.689,-7.475,-47.756,179.632,6.159,149.219
C01247=1147.694,-7.725,-47.743,179.630,6.158,149.220
C01248=1147.699,-7.974,-47.731,179.628,6.157,149.220
C01249=1147.705,-8.224,-47.717,179.625,6.157,149.221
C01250=1147.709,-8.474,-47.704,179.623,6.156,149.221
C01251=1147.714,-8.723,-47.692,179.620,6.155,149.222
C01252=1147.719,-8.972,-47.679,179.618,6.154,149.222
C01253=1147.725,-9.223,-47.666,179.615,6.154,149.223
C01254=1147.730,-9.472,-47.653,179.613,6.153,149.224
C01255=1147.735,-9.721,-47.640,179.610,6.152,149.224
C01256=1147.740,-9.971,-47.628,179.608,6.152,149.225
C01257=1147.745,-10.221,-47.615,179.606,6.151,149.225
C01258=1147.750,-10.470,-47.602,179.603,6.150,149.226
C01259=1147.756,-10.720,-47.589,179.601,6.150,149.226
C01260=1147.761,-10.969,-47.576,179.598,6.149,149.227
C01261=1147.766,-11.220,-47.564,179.596,6.147,149.228
C01262=1147.771,-11.469,-47.551,179.593,6.147,149.228
C01263=1147.777,-11.719,-47.538,179.591,6.146,149.229
C01264=1147.782,-11.968,-47.526,179.588,6.146,149.229
C01265=1147.786,-12.218,-47.513,179.586,6.145,149.230
C01266=1147.791,-12.467,-47.500,179.584,6.144,149.230
C01267=1147.796,-12.717,-47.488,179.581,6.144,149.231
C01268=1147.803,-12.967,-47.475,179.579,6.143,149.232
C01269=1147.807,-13.217,-47.462,179.576,6.143,149.232
C01270=1147.812,-13.466,-47.450,179.574,6.142,149.233
C01271=1147.817,-13.715,-47.437,179.571,6.141,149.233
C01272=1147.822,-13.965,-47.424,179.569,6.141,149.234
C01273=1147.828,-14.214,-47.412,179.566,6.139,149.235
C01274=1147.832,-14.465,-47.400,179.564,6.139,149.235
C01275=1147.838,-14.714,-47.386,179.562,6.138,149.235
C01276=1147.843,-14.964,-47.374,179.559,6.137,149.236
C01277=1147.849,-15.213,-47.361,179.557,6.136,149.237
C01278=1147.854,-15.463,-47.349,179.554,6.136,149.237
C01279=1147.859,-15.712,-47.337,179.552,6.135,149.238
C01280=1147.864,-15.962,-47.324,179.549,6.135,149.238
C01281=1147.869,-16.212,-47.311,179.547,6.134,149.239
C01282=1147.874,-16.462,-47.299,179.544,6.134,149.240
C01283=1147.879,-16.711,-47.287,179.542,6.133,149.240
C01284=1147.884,-16.960,-47.274,179.540,6.132,149.241
C01285=1147.890,-17.210,-47.262,179.537,6.132,149.241
C01286=1147.895,-17.460,-47.249,179.535,6.131,149.242
C01287=1147.900,-17.710,-47.236,179.533,6.130,149.242
C01288=1147.906,-17.960,-47.224,179.530,6.129,149.243
C01289=1147.911,-18.209,-47.211,179.527,6.128,149.244
C01290=1147.916,-18.458,-47.199,179.525,6.128,149.244
C01291=1147.921,-18.708,-47.187,179.522,6.127,149.245
C01292=1147.926,-18.958,-47.174,179.520,6.126,149.245
C01293=1147.932,-19.207,-47.162,179.518,6.126,149.246
C01294=1147.936,-19.458,-47.150,179.515,6.125,149.246
C01295=1147.942,-19.707,-47.137,179.513,6.124,149.247
C01296=1147.947,-19.957,-47.125,179.510,6.124,149.248
C01297=1147.952,-20.206,-47.112,179.508,6.123,149.248
C01298=1147.957,-20.455,-47.100,179.506,6.123,149.249
C01299=1147.963,-20.705,-47.088,179.503,6.122,149.249
C01300=1147.968,-20.955,-47.075,179.501,6.121,149.250
C01301=1147.973,-21.205,-47.063,179.499,6.121,149.250
C01302=1147.978,-21.454,-47.051,179.496,6.120,149.251
C01303=1147.984,-21.704,-47.039,179.494,6.119,149.252
C01304=1147.988,-21.954,-47.026,179.492,6.119,149.252
C01305=1147.993,-22.203,-47.013,179.489,6.118,149.253
C01306=1147.999,-22.453,-47.002,179.487,6.117,149.253
C01307=1148.004,-22.702,-46.989,179.484,6.117,149.254
C01308=1148.009,-22.952,-46.977,179.482,6.116,149.254
C01309=1148.014,-23.201,-46.965,179.480,6.115,149.255
C01310=1148.019,-23.451,-46.953,179.477,6.115,149.256
C01311=1148.024,-23.701,-46.941,179.475,6.114,149.256
C01312=1148.030,-23.951,-46.929,179.472,6.114,149.257
C01313=1148.036,-24.221,-46.915,179.470,6.113,149.257
C01314=1148.041,-24.490,-46.902,179.467,6.112,149.258
C01315=1148.047,-24.761,-46.889,179.464,6.111,149.259
C01316=1148.053,-25.030,-46.876,179.462,6.111,149.259
C01317=1148.057,-25.281,-46.864,179.459,6.110,149.260
C01318=1148.063,-25.530,-46.851,179.457,6.109,149.260
C01319=1148.068,-25.780,-46.839,179.454,6.109,149.261
C01320=1148.073,-26.030,-46.827,179.452,6.108,149.261
C01321=1148.078,-26.279,-46.816,179.450,6.107,149.262
C01322=1148.083,-26.528,-46.803,179.447,6.107,149.263
C01323=1148.088,-26.778,-46.791,179.445,6.106,149.263
C01324=1148.094,-27.028,-46.779,179.443,6.106,149.264
C01325=1148.099,-27.278,-46.767,179.440,6.105,149.264
C01326=1148.104,-27.528,-46.755,179.438,6.104,149.265
C01327=1148.109,-27.777,-46.743,179.435,6.104,149.265
C01328=1148.114,-28.027,-46.731,179.433,6.103,149.266
C01329=1148.120,-28.276,-46.719,179.431,6.102,149.267
C01330=1148.125,-28.526,-46.707,179.428,6.102,149.267
C01331=1148.130,-28.776,-46.694,179.426,6.101,149.268
C01332=1148.135,-29.025,-46.683,179.424,6.100,149.268
C01333=1148.141,-29.275,-46.672,179.421,6.100,149.269
C01334=1148.146,-29.524,-46.659,179.419,6.099,149.269
C01335=1148.151,-29.774,-46.647,179.417,6.098,149.270
C01336=1148.157,-30.024,-46.635,179.414,6.098,149.271
C01337=1148.162,-30.273,-46.624,179.412,6.097,149.271
C01338=1148.167,-30.523,-46.611,179.409,6.097,149.272
C01339=1148.172,-30.773,-46.600,179.407,6.096,149.272
C01340=1148.178,-31.023,-46.588,179.404,6.096,149.273
C01341=1148.182,-31.272,-46.576,179.402,6.095,149.273
C01342=1148.187,-31.522,-46.564,179.399,6.094,149.274
C01343=1148.193,-31.771,-46.552,179.397,6.094,149.274
C01344=1148.198,-32.021,-46.540,179.395,6.093,149.275
C01345=1148.203,-32.271,-46.529,179.392,6.092,149.276
C01346=1148.208,-32.520,-46.516,179.390,6.092,149.276
C01347=1148.213,-32.770,-46.504,179.388,6.091,149.277
C01348=1148.218,-33.020,-46.493,179.385,6.090,149.277
C01349=1148.224,-33.269,-46.481,179.383,6.090,149.278
C01350=1148.230,-33.519,-46.470,179.381,6.090,149.278
C01351=1148.234,-33.769,-46.458,179.379,6.089,149.279
C01352=1148.239,-34.018,-46.446,179.376,6.089,149.280
C01353=1148.245,-34.268,-46.434,179.374,6.088,149.280
C01354=1148.250,-34.518,-46.422,179.371,6.088,149.281
C01355=1148.255,-34.768,-46.411,179.369,6.087,149.281
C01356=1148.260,-35.017,-46.399,179.367,6.086,149.282
C01357=1148.266,-35.267,-46.387,179.364,6.086,149.282
C01358=1148.271,-35.516,-46.376,179.362,6.085,149.283
C01359=1148.277,-35.766,-46.364,179.359,6.084,149.284
C01360=1148.281,-36.016,-46.353,179.357,6.084,149.284
C01361=1148.286,-36.265,-46.340,179.355,6.083,149.285
C01362=1148.292,-36.515,-46.328,179.352,6.082,149.285
C01363=1148.297,-36.765,-46.317,179.350,6.082,149.286
C01364=1148.303,-37.014,-46.305,179.348,6.081,149.286
C01365=1148.308,-37.264,-46.294,179.345,6.080,149.287
C01366=1148.313,-37.514,-46.282,179.343,6.080,149.288
C01367=1148.318,-37.764,-46.270,179.341,6.079,149.288
C01368=1148.323,-38.013,-46.259,179.338,6.079,149.289
C01369=1148.328,-38.263,-46.247,179.336,6.079,149.289
C01370=1148.334,-38.512,-46.236,179.334,6.078,149.290
C01371=1148.339,-38.762,-46.224,179.331,6.078,149.290
C01372=1148.344,-39.012,-46.212,179.329,6.077,149.291
C01373=1148.349,-39.261,-46.201,179.327,6.076,149.292
C01374=1148.354,-39.511,-46.189,179.324,6.076,149.292
C01375=1148.360,-39.760,-46.178,179.322,6.075,149.293
C01376=1148.365,-40.010,-46.166,179.320,6.074,149.293
C01377=1148.371,-40.260,-46.155,179.317,6.074,149.294
C01378=1148.375,-40.510,-46.143,179.315,6.073,149.294
C01379=1148.381,-40.760,-46.131,179.313,6.073,149.295
C01380=1148.386,-41.009,-46.120,179.310,6.072,149.295
C01381=1148.391,-41.259,-46.109,179.308,6.071,149.296
C01382=1148.396,-41.509,-46.098,179.306,6.071,149.297
C01383=1148.402,-41.759,-46.086,179.303,6.071,149.297
C01384=1148.407,-42.008,-46.075,179.301,6.070,149.298
C01385=1148.413,-42.258,-46.063,179.299,6.070,149.298
C01386=1148.417,-42.507,-46.052,179.296,6.069,149.299
C01387=1148.423,-42.757,-46.040,179.294,6.068,149.299
C01388=1148.427,-43.007,-46.029,179.292,6.068,149.300
C01389=1148.433,-43.256,-46.017,179.289,6.067,149.301
C01390=1148.438,-43.506,-46.006,179.287,6.067,149.301
C01391=1148.444,-43.756,-45.995,179.285,6.066,149.302
C01392=1148.449,-44.006,-45.984,179.282,6.065,149.302
C01393=1148.455,-44.255,-45.972,179.280,6.065,149.303
C01394=1148.459,-44.505,-45.961,179.278,6.065,149.303
C01395=1148.464,-44.754,-45.950,179.275,6.064,149.304
C01396=1148.469,-45.004,-45.938,179.273,6.063,149.305
C01397=1148.475,-45.254,-45.927,179.271,6.063,149.305
C01398=1148.480,-45.504,-45.916,179.268,6.062,149.306
C01399=1148.485,-45.753,-45.904,179.266,6.061,149.306
C01400=1148.491,-46.003,-45.893,179.264,6.061,149.307
C01401=1148.496,-46.253,-45.882,179.261,6.060,149.307
C01402=1148.501,-46.503,-45.871,179.259,6.059,149.308
C01403=1148.506,-46.752,-45.859,179.257,6.060,149.309
C01404=1148.512,-47.001,-45.848,179.255,6.059,149.309
C01405=1148.517,-47.252,-45.837,179.252,6.059,149.310
C01406=1148.522,-47.502,-45.826,179.250,6.058,149.310
C01407=1148.527,-47.751,-45.815,179.248,6.057,149.311
C01408=1148.533,-48.000,-45.803,179.245,6.057,149.311
C01409=1148.538,-48.251,-45.792,179.243,6.056,149.312
C01410=1148.543,-48.500,-45.781,179.240,6.056,149.313
C01411=1148.548,-48.750,-45.769,179.239,6.056,149.313
C01412=1148.553,-49.000,-45.759,179.237,6.055,149.314
C01413=1148.559,-49.249,-45.747,179.234,6.054,149.314
C01414=1148.564,-49.499,-45.736,179.232,6.054,149.315
C01415=1148.569,-49.749,-45.725,179.229,6.053,149.315
C01416=1148.575,-49.998,-45.714,179.227,6.052,149.316
C01417=1148.580,-50.269,-45.702,179.224,6.052,149.317
C01418=1148.586,-50.540,-45.690,179.222,6.051,149.317
C01419=1148.592,-50.810,-45.678,179.219,6.051,149.318
C01420=1148.598,-51.081,-45.666,179.217,6.050,149.318
C01421=1148.603,-51.330,-45.655,179.214,6.050,149.319
C01422=1148.608,-51.580,-45.644,179.212,6.049,149.320
C01423=1148.613,-51.830,-45.632,179.210,6.049,149.320
C01424=1148.619,-52.079,-45.622,179.208,6.048,149.321
C01425=1148.624,-52.329,-45.611,179.206,6.048,149.321
C01426=1148.628,-52.579,-45.600,179.203,6.047,149.322
C01427=1148.635,-52.829,-45.589,179.201,6.046,149.322
C01428=1148.639,-53.078,-45.578,179.198,6.046,149.323
C01429=1148.645,-53.327,-45.567,179.196,6.045,149.324
C01430=1148.650,-53.578,-45.556,179.195,6.045,149.324
C01431=1148.655,-53.828,-45.544,179.192,6.045,149.325
C01432=1148.661,-54.077,-45.534,179.190,6.044,149.325
C01433=1148.665,-54.327,-45.523,179.187,6.044,149.326
C01434=1148.671,-54.576,-45.513,179.185,6.043,149.326
C01435=1148.676,-54.826,-45.501,179.183,6.042,149.327
C01436=1148.681,-55.076,-45.490,179.181,6.043,149.328
C01437=1148.687,-55.325,-45.479,179.178,6.042,149.328
C01438=1148.692,-55.576,-45.469,179.176,6.041,149.329
C01439=1148.697,-55.825,-45.458,179.174,6.041,149.329
C01440=1148.703,-56.075,-45.446,179.171,6.040,149.330
C01441=1148.707,-56.325,-45.435,179.169,6.039,149.330
C01442=1148.713,-56.574,-45.425,179.166,6.039,149.331
C01443=1148.718,-56.824,-45.414,179.165,6.039,149.331
C01444=1148.723,-57.073,-45.403,179.162,6.038,149.332
C01445=1148.729,-57.323,-45.392,179.160,6.038,149.333
C01446=1148.734,-57.573,-45.381,179.158,6.037,149.333
C01447=1148.739,-57.823,-45.371,179.155,6.036,149.334
C01448=1148.745,-58.072,-45.360,179.154,6.036,149.334
C01449=1148.750,-58.322,-45.349,179.151,6.036,149.335
C01450=1148.755,-58.571,-45.338,179.149,6.035,149.335
C01451=1148.760,-58.821,-45.328,179.147,6.034,149.336
C01452=1148.766,-59.072,-45.317,179.144,6.034,149.337
C01453=1148.771,-59.321,-45.306,179.142,6.033,149.337
C01454=1148.776,-59.571,-45.295,179.140,6.033,149.338
C01455=1148.781,-59.820,-45.284,179.137,6.033,149.338
C01456=1148.786,-60.070,-45.274,179.135,6.032,149.339
C01457=1148.792,-60.320,-45.263,179.133,6.032,149.339
C01458=1148.796,-60.570,-45.252,179.130,6.031,149.340
C01459=1148.802,-60.819,-45.242,179.129,6.031,149.340
C01460=1148.807,-61.069,-45.231,179.126,6.031,149.341
C01461=1148.812,-61.318,-45.220,179.124,6.030,149.342
C01462=1148.818,-61.569,-45.209,179.122,6.029,149.342
C01463=1148.824,-61.818,-45.199,179.119,6.029,149.343
C01464=1148.828,-62.068,-45.188,179.117,6.029,149.343
C01465=1148.834,-62.318,-45.178,179.115,6.028,149.344
C01466=1148.839,-62.568,-45.167,179.113,6.027,149.344
C01467=1148.845,-62.817,-45.157,179.110,6.027,149.345
C01468=1148.849,-63.067,-45.145,179.108,6.026,149.346
C01469=1148.855,-63.316,-45.135,179.106,6.026,149.346
C01470=1148.860,-63.566,-45.125,179.104,6.026,149.347
C01471=1148.865,-63.816,-45.114,179.101,6.025,149.347
C01472=1148.871,-64.065,-45.104,179.099,6.024,149.348
C01473=1148.876,-64.315,-45.093,179.097,6.024,149.348
C01474=1148.881,-64.565,-45.083,179.095,6.024,149.349
C01475=1148.886,-64.815,-45.072,179.093,6.023,149.349
C01476=1148.892,-65.064,-45.061,179.090,6.023,149.350
C01477=1148.897,-65.314,-45.051,179.088,6.022,149.351
C01478=1148.902,-65.564,-45.040,179.086,6.021,149.351
C01479=1148.908,-65.813,-45.030,179.084,6.022,149.352
C01480=1148.913,-66.064,-45.020,179.081,6.021,149.352
C01481=1148.918,-66.313,-45.009,179.079,6.020,149.353
C01482=1148.923,-66.563,-44.998,179.076,6.020,149.353
C01483=1148.929,-66.812,-44.988,179.074,6.019,149.354
C01484=1148.934,-67.063,-44.977,179.073,6.019,149.354
C01485=1148.939,-67.312,-44.967,179.070,6.019,149.355
C01486=1148.945,-67.562,-44.957,179.068,6.018,149.356
C01487=1148.950,-67.812,-44.946,179.066,6.017,149.356
C01488=1148.955,-68.061,-44.936,179.064,6.017,149.357
C01489=1148.960,-68.311,-44.925,179.061,6.017,149.357
C01490=1148.966,-68.561,-44.915,179.059,6.016,149.358
C01491=1148.971,-68.810,-44.905,179.057,6.016,149.358
C01492=1148.976,-69.061,-44.894,179.055,6.016,149.359
C01493=1148.981,-69.310,-44.884,179.053,6.015,149.359
C01494=1148.987,-69.559,-44.874,179.050,6.014,149.360
C01495=1148.992,-69.810,-44.864,179.048,6.014,149.361
C01496=1148.997,-70.059,-44.853,179.045,6.013,149.361
C01497=1149.002,-70.309,-44.843,179.044,6.013,149.362
C01498=1149.008,-70.559,-44.833,179.041,6.012,149.362
C01499=1149.014,-70.808,-44.822,179.039,6.012,149.363
C01500=1149.019,-71.059,-44.812,179.037,6.011,149.363
C01501=1149.024,-71.308,-44.801,179.035,6.011,149.364
C01502=1149.029,-71.557,-44.791,179.032,6.011,149.365
C01503=1149.034,-71.807,-44.781,179.030,6.010,149.365
C01504=1149.039,-72.057,-44.770,179.028,6.009,149.366
C01505=1149.045,-72.306,-44.760,179.026,6.010,149.366
C01506=1149.050,-72.556,-44.750,179.024,6.009,149.367
C01507=1149.056,-72.806,-44.739,179.021,6.008,149.367
C01508=1149.061,-73.055,-44.729,179.019,6.008,149.368
C01509=1149.066,-73.306,-44.719,179.017,6.008,149.368
C01510=1149.071,-73.556,-44.710,179.015,6.007,149.369
C01511=1149.077,-73.805,-44.700,179.012,6.007,149.370
C01512=1149.082,-74.055,-44.689,179.010,6.006,149.370
C01513=1149.087,-74.305,-44.679,179.009,6.006,149.371
C01514=1149.093,-74.554,-44.669,179.006,6.006,149.371
C01515=1149.099,-74.804,-44.658,179.004,6.005,149.372
C01516=1149.103,-75.054,-44.648,179.002,6.005,149.372
C01517=1149.109,-75.303,-44.638,178.999,6.005,149.373
C01518=1149.114,-75.553,-44.628,178.997,6.004,149.374
C01519=1149.119,-75.803,-44.617,178.995,6.003,149.374
C01520=1149.125,-76.053,-44.607,178.993,6.003,149.374
C01521=1149.131,-76.323,-44.597,178.991,6.003,149.375
C01522=1149.137,-76.596,-44.586,178.988,6.002,149.376
C01523=1149.142,-76.867,-44.575,178.986,6.001,149.376
C01524=1149.148,-77.139,-44.563,178.983,6.001,149.377
C01525=1149.153,-77.388,-44.554,178.981,6.000,149.378
C01526=1149.158,-77.637,-44.544,178.979,6.000,149.378
C01527=1149.164,-77.887,-44.534,178.977,6.000,149.379
C01528=1149.169,-78.138,-44.523,178.975,5.999,149.379
C01529=1149.174,-78.387,-44.514,178.972,5.998,149.380
C01530=1149.180,-78.636,-44.504,178.971,5.998,149.380
C01531=1149.185,-78.886,-44.493,178.968,5.998,149.381
C01532=1149.190,-79.136,-44.483,178.966,5.997,149.381
C01533=1149.195,-79.386,-44.474,178.964,5.997,149.382
C01534=1149.201,-79.636,-44.464,178.962,5.997,149.383
C01535=1149.207,-79.885,-44.454,178.959,5.996,149.383
C01536=1149.212,-80.134,-44.444,178.957,5.995,149.384
C01537=1149.217,-80.385,-44.433,178.955,5.996,149.384
C01538=1149.222,-80.635,-44.424,178.953,5.995,149.385
C01539=1149.227,-80.884,-44.414,178.951,5.994,149.385
C01540=1149.233,-81.134,-44.404,178.949,5.995,149.386
C01541=1149.238,-81.384,-44.393,178.947,5.994,149.386
C01542=1149.243,-81.634,-44.385,178.944,5.993,149.387
C01543=1149.249,-81.883,-44.374,178.943,5.993,149.387
C01544=1149.254,-82.133,-44.364,178.940,5.993,149.388
C01545=1149.259,-82.382,-44.355,178.938,5.992,149.389
C01546=1149.264,-82.633,-44.345,178.936,5.991,149.389
C01547=1149.270,-82.882,-44.334,178.934,5.992,149.390
C01548=1149.275,-83.132,-44.325,178.931,5.991,149.390
C01549=1149.281,-83.382,-44.315,178.929,5.990,149.391
C01550=1149.286,-83.631,-44.305,178.927,5.991,149.391
C01551=1149.291,-83.881,-44.296,178.925,5.990,149.392
C01552=1149.297,-84.131,-44.286,178.923,5.989,149.392
C01553=1149.302,-84.381,-44.275,178.921,5.989,149.393
C01554=1149.307,-84.630,-44.266,178.919,5.989,149.394
C01555=1149.313,-84.880,-44.256,178.916,5.988,149.394
C01556=1149.318,-85.130,-44.247,178.914,5.987,149.395
C01557=1149.323,-85.380,-44.236,178.912,5.988,149.395
C01558=1149.328,-85.630,-44.227,178.910,5.987,149.396
C01559=1149.334,-85.879,-44.217,178.908,5.986,149.396
C01560=1149.339,-86.129,-44.207,178.906,5.986,149.397
C01561=1149.344,-86.379,-44.198,178.903,5.986,149.397
C01562=1149.350,-86.628,-44.188,178.901,5.985,149.398
C01563=1149.355,-86.878,-44.179,178.900,5.985,149.398
C01564=1149.360,-87.128,-44.168,178.897,5.985,149.399
C01565=1149.365,-87.378,-44.159,178.895,5.984,149.400
C01566=1149.371,-87.628,-44.149,178.893,5.984,149.400
C01567=1149.376,-87.877,-44.139,178.891,5.983,149.401
C01568=1149.382,-88.127,-44.130,178.888,5.983,149.401
C01569=1149.387,-88.377,-44.120,178.887,5.983,149.402
C01570=1149.392,-88.626,-44.111,178.884,5.982,149.402
C01571=1149.398,-88.876,-44.101,178.882,5.982,149.403
C01572=1149.402,-89.127,-44.091,178.880,5.982,149.403
C01573=1149.408,-89.376,-44.081,178.878,5.981,149.404
C01574=1149.413,-89.626,-44.072,178.876,5.980,149.404
C01575=1149.419,-89.876,-44.062,178.874,5.981,149.405
C01576=1149.424,-90.125,-44.053,178.872,5.980,149.406
C01577=1149.430,-90.375,-44.043,178.869,5.979,149.406
C01578=1149.434,-90.624,-44.033,178.868,5.979,149.407
C01579=1149.440,-90.874,-44.024,178.865,5.979,149.407
C01580=1149.446,-91.124,-44.015,178.863,5.978,149.408
C01581=1149.451,-91.374,-44.005,178.861,5.978,149.408
C01582=1149.456,-91.624,-43.996,178.859,5.977,149.409
C01583=1149.461,-91.874,-43.985,178.856,5.977,149.409
C01584=1149.466,-92.124,-43.976,178.855,5.977,149.410
C01585=1149.471,-92.373,-43.967,178.853,5.976,149.410
C01586=1149.477,-92.623,-43.957,178.850,5.976,149.411
C01587=1149.482,-92.872,-43.948,178.848,5.976,149.412
C01588=1149.488,-93.122,-43.938,178.846,5.975,149.412
C01589=1149.493,-93.372,-43.929,178.844,5.974,149.413
C01590=1149.499,-93.622,-43.919,178.842,5.975,149.413
C01591=1149.504,-93.872,-43.910,178.840,5.974,149.414
C01592=1149.510,-94.121,-43.900,178.838,5.974,149.414
C01593=1149.515,-94.371,-43.891,178.836,5.973,149.415
C01594=1149.520,-94.620,-43.882,178.833,5.973,149.415
C01595=1149.525,-94.870,-43.872,178.832,5.973,149.416
C01596=1149.531,-95.120,-43.863,178.829,5.972,149.416
C01597=1149.536,-95.370,-43.853,178.827,5.971,149.417
C01598=1149.541,-95.620,-43.844,178.825,5.972,149.418
C01599=1149.547,-95.870,-43.835,178.823,5.971,149.418
C01600=1149.552,-96.119,-43.825,178.821,5.970,149.419
C01601=1149.557,-96.369,-43.816,178.819,5.970,149.419
C01602=1149.563,-96.619,-43.807,178.817,5.970,149.420
C01603=1149.568,-96.868,-43.797,178.815,5.970,149.420
C01604=1149.573,-97.118,-43.788,178.813,5.969,149.421
C01605=1149.579,-97.368,-43.779,178.811,5.968,149.421
C01606=1149.584,-97.618,-43.769,178.808,5.969,149.422
C01607=1149.589,-97.867,-43.760,178.806,5.968,149.422
C01608=1149.595,-98.118,-43.751,178.804,5.967,149.423
C01609=1149.600,-98.367,-43.741,178.803,5.967,149.423
C01610=1149.605,-98.617,-43.732,178.800,5.966,149.424
C01611=1149.611,-98.867,-43.723,178.798,5.967,149.425
C01612=1149.616,-99.117,-43.714,178.796,5.966,149.425
C01613=1149.621,-99.366,-43.704,178.794,5.965,149.426
C01614=1149.627,-99.616,-43.695,178.792,5.965,149.426
C01615=1149.632,-99.866,-43.686,178.790,5.965,149.427
C01616=1149.637,-100.116,-43.677,178.787,5.964,149.427
C01617=1149.643,-100.365,-43.666,178.786,5.964,149.428
C01618=1149.648,-100.615,-43.658,178.784,5.964,149.428
C01619=1149.653,-100.865,-43.649,178.782,5.964,149.429
C01620=1149.659,-101.115,-43.639,178.779,5.963,149.429
C01621=1149.664,-101.365,-43.630,178.777,5.962,149.430
C01622=1149.669,-101.614,-43.621,178.776,5.963,149.430
C01623=1149.674,-101.864,-43.612,178.773,5.962,149.431
C01624=1149.680,-102.114,-43.602,178.771,5.962,149.432
C01625=1149.686,-102.386,-43.592,178.769,5.961,149.432
C01626=1149.692,-102.658,-43.583,178.767,5.961,149.433
C01627=1149.698,-102.930,-43.573,178.764,5.960,149.433
C01628=1149.703,-103.203,-43.563,178.763,5.960,149.434
C01629=1149.708,-103.452,-43.554,178.760,5.960,149.434
C01630=1149.714,-103.702,-43.544,178.758,5.959,149.435
C01631=1149.719,-103.952,-43.535,178.756,5.959,149.435
C01632=1149.725,-104.202,-43.526,178.754,5.958,149.436
C01633=1149.730,-104.451,-43.518,178.752,5.959,149.436
C01634=1149.736,-104.701,-43.508,178.750,5.958,149.437
C01635=1149.741,-104.951,-43.499,178.747,5.957,149.438
C01636=1149.746,-105.200,-43.490,178.746,5.957,149.438
C01637=1149.751,-105.450,-43.481,178.744,5.957,149.439
C01638=1149.757,-105.700,-43.472,178.742,5.957,149.439
C01639=1149.762,-105.950,-43.462,178.740,5.956,149.440
C01640=1149.768,-106.200,-43.454,178.737,5.956,149.440
C01641=1149.773,-106.450,-43.445,178.736,5.956,149.441
C01642=1149.779,-106.699,-43.436,178.733,5.955,149.441
C01643=1149.784,-106.949,-43.427,178.732,5.955,149.442
C01644=1149.789,-107.198,-43.418,178.730,5.954,149.442
C01645=1149.795,-107.449,-43.409,178.727,5.954,149.443
C01646=1149.800,-107.698,-43.400,178.725,5.954,149.443
C01647=1149.805,-107.948,-43.391,178.723,5.953,149.444
C01648=1149.810,-108.198,-43.382,178.722,5.953,149.444
C01649=1149.815,-108.448,-43.373,178.719,5.952,149.445
C01650=1149.821,-108.697,-43.365,178.717,5.953,149.446
C01651=1149.827,-108.947,-43.355,178.715,5.952,149.446
C01652=1149.832,-109.197,-43.346,178.713,5.951,149.447
C01653=1149.837,-109.447,-43.337,178.711,5.951,149.447
C01654=1149.843,-109.697,-43.329,178.709,5.951,149.448
C01655=1149.848,-109.947,-43.320,178.707,5.951,149.448
C01656=1149.854,-110.196,-43.311,178.705,5.950,149.449
C01657=1149.859,-110.446,-43.302,178.703,5.950,149.449
C01658=1149.864,-110.696,-43.293,178.701,5.950,149.450
C01659=1149.870,-110.946,-43.284,178.699,5.949,149.450
C01660=1149.875,-111.196,-43.275,178.697,5.949,149.451
C01661=1149.880,-111.445,-43.266,178.695,5.948,149.451
C01662=1149.886,-111.695,-43.257,178.693,5.948,149.452
C01663=1149.891,-111.944,-43.249,178.691,5.948,149.452
C01664=1149.896,-112.194,-43.240,178.689,5.948,149.453
C01665=1149.901,-112.444,-43.231,178.687,5.947,149.453
C01666=1149.907,-112.694,-43.222,178.685,5.946,149.454
C01667=1149.912,-112.943,-43.213,178.683,5.947,149.455
C01668=1149.917,-113.193,-43.204,178.680,5.946,149.455
C01669=1149.923,-113.444,-43.196,178.679,5.946,149.456
C01670=1149.928,-113.693,-43.187,178.677,5.945,149.456
C01671=1149.933,-113.943,-43.178,178.675,5.945,149.457
C01672=1149.939,-114.192,-43.170,178.673,5.944,149.457
C01673=1149.945,-114.443,-43.160,178.671,5.945,149.458
C01674=1149.950,-114.692,-43.152,178.669,5.944,149.458
C01675=1149.955,-114.942,-43.143,178.666,5.943,149.459
C01676=1149.961,-115.191,-43.134,178.665,5.943,149.459
C01677=1149.967,-115.442,-43.126,178.663,5.943,149.460
C01678=1149.972,-115.692,-43.117,178.661,5.943,149.460
C01679=1149.977,-115.942,-43.108,178.659,5.942,149.461
C01680=1149.983,-116.191,-43.100,178.657,5.942,149.461
C01681=1149.988,-116.441,-43.091,178.655,5.942,149.462
C01682=1149.993,-116.690,-43.082,178.653,5.942,149.462
C01683=1149.998,-116.941,-43.074,178.651,5.941,149.463
C01684=1150.004,-117.190,-43.065,178.649,5.941,149.463
C01685=1150.009,-117.440,-43.056,178.647,5.940,149.464
C01686=1150.015,-117.690,-43.047,178.645,5.939,149.464
C01687=1150.020,-117.940,-43.039,178.643,5.940,149.465
C01688=1150.026,-118.189,-43.031,178.641,5.939,149.465
C01689=1150.031,-118.439,-43.022,178.639,5.939,149.466
C01690=1150.036,-118.689,-43.013,178.637,5.938,149.466
C01691=1150.041,-118.939,-43.004,178.635,5.938,149.467
C01692=1150.047,-119.188,-42.997,178.633,5.938,149.467
C01693=1150.052,-119.438,-42.988,178.631,5.938,149.468
C01694=1150.057,-119.688,-42.979,178.629,5.937,149.469
C01695=1150.063,-119.937,-42.970,178.627,5.937,149.469
C01696=1150.068,-120.188,-42.962,178.625,5.937,149.470
C01697=1150.073,-120.438,-42.953,178.623,5.937,149.470
C01698=1150.079,-120.687,-42.944,178.621,5.936,149.471
C01699=1150.085,-120.937,-42.937,178.619,5.936,149.471
C01700=1150.090,-121.187,-42.928,178.617,5.935,149.472
C01701=1150.095,-121.437,-42.919,178.615,5.935,149.472
C01702=1150.101,-121.687,-42.911,178.613,5.935,149.473
C01703=1150.106,-121.936,-42.902,178.611,5.934,149.473
C01704=1150.111,-122.186,-42.894,178.609,5.934,149.474
C01705=1150.117,-122.436,-42.886,178.607,5.934,149.474
C01706=1150.122,-122.686,-42.877,178.605,5.934,149.475
C01707=1150.127,-122.935,-42.868,178.603,5.933,149.475
C01708=1150.133,-123.185,-42.860,178.602,5.933,149.476
C01709=1150.138,-123.435,-42.851,178.599,5.932,149.476
C01710=1150.143,-123.685,-42.843,178.598,5.932,149.477
C01711=1150.149,-123.935,-42.835,178.596,5.931,149.477
C01712=1150.154,-124.184,-42.826,178.594,5.932,149.478
C01713=1150.159,-124.434,-42.818,178.591,5.931,149.478
C01714=1150.165,-124.684,-42.810,178.590,5.931,149.479
C01715=1150.170,-124.934,-42.801,178.588,5.930,149.479
C01716=1150.176,-125.184,-42.793,178.586,5.930,149.480
C01717=1150.182,-125.433,-42.784,178.584,5.930,149.480
C01718=1150.187,-125.683,-42.775,178.582,5.930,149.481
C01719=1150.191,-125.933,-42.768,178.580,5.929,149.481
C01720=1150.197,-126.183,-42.759,178.578,5.929,149.482
C01721=1150.203,-126.433,-42.751,178.576,5.928,149.482
C01722=1150.208,-126.682,-42.742,178.574,5.929,149.483
C01723=1150.214,-126.933,-42.734,178.572,5.928,149.483
C01724=1150.218,-127.182,-42.726,178.570,5.928,149.484
C01725=1150.224,-127.431,-42.717,178.568,5.927,149.484
C01726=1150.230,-127.682,-42.709,178.567,5.927,149.485
C01727=1150.235,-127.932,-42.700,178.564,5.927,149.485
C01728=1150.241,-128.181,-42.692,178.563,5.927,149.486
C01729=1149.820,-128.193,-42.735,178.559,5.930,149.488
C01730=1149.814,-127.942,-42.743,178.561,5.931,149.487
C01731=1149.809,-127.693,-42.752,178.563,5.931,149.487
C01732=1149.803,-127.443,-42.760,178.565,5.931,149.486
C01733=1149.798,-127.193,-42.769,178.567,5.931,149.486
C01734=1149.793,-126.944,-42.777,178.569,5.932,149.485
C01735=1149.787,-126.694,-42.785,178.571,5.932,149.485
C01736=1149.782,-126.444,-42.794,178.573,5.932,149.484
C01737=1149.776,-126.194,-42.802,178.575,5.932,149.484
C01738=1149.771,-125.944,-42.810,178.577,5.933,149.483
C01739=1149.765,-125.694,-42.819,178.578,5.933,149.483
C01740=1149.760,-125.445,-42.827,178.581,5.934,149.482
C01741=1149.755,-125.195,-42.835,178.582,5.934,149.482
C01742=1149.749,-124.945,-42.843,178.584,5.934,149.481
C01743=1149.744,-124.695,-42.852,178.586,5.934,149.481
C01744=1149.738,-124.445,-42.860,178.589,5.935,149.480
C01745=1149.733,-124.196,-42.869,178.590,5.935,149.479
C01746=1149.728,-123.946,-42.877,178.592,5.935,149.479
C01747=1149.723,-123.696,-42.885,178.594,5.935,149.478
C01748=1149.717,-123.447,-42.894,178.596,5.936,149.478
C01749=1149.712,-123.196,-42.902,178.598,5.936,149.477
C01750=1149.706,-122.946,-42.911,178.600,5.937,149.477
C01751=1149.701,-122.697,-42.919,178.602,5.937,149.477
C01752=1149.695,-122.447,-42.928,178.604,5.938,149.476
C01753=1149.690,-122.197,-42.937,178.605,5.938,149.476
C01754=1149.685,-121.948,-42.945,178.608,5.938,149.475
C01755=1149.679,-121.697,-42.953,178.610,5.938,149.474
C01756=1149.674,-121.448,-42.962,178.612,5.939,149.474
C01757=1149.669,-121.198,-42.970,178.613,5.939,149.473
C01758=1149.663,-120.949,-42.979,178.616,5.939,149.473
C01759=1149.658,-120.698,-42.987,178.617,5.939,149.472
C01760=1149.653,-120.448,-42.996,178.619,5.940,149.472
C01761=1149.647,-120.199,-43.005,178.622,5.941,149.471
C01762=1149.641,-119.949,-43.013,178.623,5.941,149.471
C01763=1149.636,-119.699,-43.022,178.626,5.941,149.470
C01764=1149.631,-119.450,-43.030,178.627,5.941,149.470
C01765=1149.625,-119.200,-43.039,178.630,5.942,149.469
C01766=1149.621,-118.950,-43.047,178.631,5.942,149.469
C01767=1149.615,-118.700,-43.056,178.633,5.942,149.468
C01768=1149.610,-118.451,-43.064,178.635,5.942,149.468
C01769=1149.605,-118.201,-43.073,178.637,5.943,149.467
C01770=1149.599,-117.950,-43.081,178.639,5.943,149.467
C01771=1149.594,-117.701,-43.090,178.642,5.944,149.466
C01772=1149.588,-117.451,-43.099,178.643,5.943,149.466
C01773=1149.583,-117.202,-43.108,178.645,5.944,149.465
C01774=1149.578,-116.952,-43.116,178.648,5.945,149.465
C01775=1149.572,-116.702,-43.124,178.649,5.945,149.464
C01776=1149.567,-116.452,-43.133,178.651,5.946,149.464
C01777=1149.561,-116.202,-43.142,178.653,5.946,149.463
C01778=1149.556,-115.952,-43.151,178.656,5.946,149.462
C01779=1149.550,-115.703,-43.160,178.657,5.946,149.462
C01780=1149.545,-115.453,-43.168,178.659,5.947,149.461
C01781=1149.540,-115.203,-43.177,178.661,5.947,149.461
C01782=1149.535,-114.953,-43.185,178.663,5.947,149.461
C01783=1149.529,-114.703,-43.194,178.665,5.947,149.460
C01784=1149.524,-114.454,-43.203,178.667,5.948,149.460
C01785=1149.519,-114.204,-43.212,178.670,5.949,149.459
C01786=1149.513,-113.954,-43.221,178.671,5.948,149.458
C01787=1149.507,-113.704,-43.229,178.673,5.949,149.458
C01788=1149.501,-113.454,-43.238,178.675,5.949,149.457
C01789=1149.496,-113.205,-43.247,178.677,5.950,149.457
C01790=1149.491,-112.955,-43.256,178.679,5.950,149.456
C01791=1149.486,-112.705,-43.265,178.682,5.950,149.456
C01792=1149.481,-112.455,-43.274,178.683,5.950,149.455
C01793=1149.475,-112.206,-43.282,178.685,5.951,149.455
C01794=1149.470,-111.956,-43.291,178.688,5.952,149.454
C01795=1149.465,-111.706,-43.300,178.689,5.952,149.454
C01796=1149.459,-111.456,-43.309,178.691,5.952,149.453
C01797=1149.454,-111.206,-43.318,178.693,5.952,149.453
C01798=1149.449,-110.957,-43.326,178.696,5.953,149.452
C01799=1149.443,-110.707,-43.334,178.697,5.953,149.452
C01800=1149.437,-110.457,-43.344,178.699,5.954,149.451
C01801=1149.432,-110.207,-43.353,178.702,5.954,149.451
C01802=1149.427,-109.957,-43.362,178.703,5.954,149.450
C01803=1149.422,-109.707,-43.371,178.706,5.955,149.449
C01804=1149.416,-109.458,-43.379,178.707,5.955,149.449
C01805=1149.411,-109.208,-43.388,178.710,5.955,149.448
C01806=1149.406,-108.958,-43.397,178.711,5.955,149.448
C01807=1149.400,-108.708,-43.406,178.713,5.956,149.447
C01808=1149.394,-108.458,-43.415,178.716,5.957,149.447
C01809=1149.389,-108.208,-43.424,178.718,5.956,149.446
C01810=1149.384,-107.959,-43.433,178.720,5.957,149.446
C01811=1149.378,-107.709,-43.442,178.721,5.957,149.445
C01812=1149.373,-107.460,-43.451,178.724,5.958,149.445
C01813=1149.368,-107.210,-43.460,178.726,5.959,149.444
C01814=1149.362,-106.960,-43.470,178.728,5.958,149.444
C01815=1149.357,-106.710,-43.479,178.730,5.959,149.443
C01816=1149.352,-106.460,-43.487,178.732,5.959,149.443
C01817=1149.347,-106.211,-43.496,178.734,5.960,149.442
C01818=1149.341,-105.961,-43.505,178.736,5.960,149.442
C01819=1149.336,-105.712,-43.514,178.738,5.960,149.441
C01820=1149.330,-105.461,-43.523,178.740,5.961,149.440
C01821=1149.325,-105.212,-43.532,178.742,5.961,149.440
C01822=1149.320,-104.962,-43.541,178.744,5.961,149.439
C01823=1149.315,-104.712,-43.550,178.746,5.961,149.439
C01824=1149.309,-104.462,-43.559,178.748,5.962,149.438
C01825=1149.304,-104.212,-43.569,178.751,5.963,149.438
C01826=1149.299,-103.963,-43.578,178.752,5.962,149.437
C01827=1149.294,-103.713,-43.587,178.754,5.963,149.437
